LIN {X 0.120,Y -564.110,Z 895.304,A 0.000,B 0.000,C 90.000,E1 90.630} C_DIS
LIN {X 0.098,Y -564.403,Z 895.296,A 0.000,B 0.000,C 90.000,E1 89.255} C_DIS
LIN {X 0.202,Y -564.749,Z 895.287,A 0.000,B 0.000,C 90.000,E1 87.593} C_DIS
LIN {X -0.113,Y -565.091,Z 895.276,A 0.000,B 0.000,C 90.000,E1 85.698} C_DIS
LIN {X 0.186,Y -565.411,Z 895.265,A 0.000,B 0.000,C 90.000,E1 83.742} C_DIS
LIN {X -0.178,Y -565.787,Z 895.256,A 0.000,B 0.000,C 90.000,E1 82.129} C_DIS
LIN {X -0.129,Y -566.486,Z 895.244,A 0.000,B 0.000,C 90.000,E1 79.926} C_DIS
LIN {X -0.025,Y -567.332,Z 895.233,A 0.000,B 0.000,C 90.000,E1 77.993} C_DIS
LIN {X -0.074,Y -568.104,Z 895.224,A 0.000,B 0.000,C 90.000,E1 76.353} C_DIS
LIN {X -0.157,Y -568.803,Z 895.217,A 0.000,B 0.000,C 90.000,E1 74.991} C_DIS
LIN {X -0.072,Y -569.345,Z 895.209,A 0.000,B 0.000,C 90.000,E1 73.614} C_DIS
LIN {X 0.196,Y -569.893,Z 895.200,A 0.000,B 0.000,C 90.000,E1 71.945} C_DIS
LIN {X -0.062,Y -570.251,Z 895.192,A 0.000,B 0.000,C 90.000,E1 70.604} C_DIS
LIN {X -0.125,Y -570.430,Z 895.186,A 0.000,B 0.000,C 90.000,E1 69.518} C_DIS
LIN {X 0.185,Y -570.675,Z 895.177,A 0.000,B 0.000,C 90.000,E1 67.847} C_DIS
LIN {X -0.023,Y -570.852,Z 895.168,A 0.000,B 0.000,C 90.000,E1 66.230} C_DIS
LIN {X 0.003,Y -570.849,Z 895.159,A 0.000,B 0.000,C 90.000,E1 64.588} C_DIS
LIN {X 0.188,Y -570.834,Z 895.151,A 0.000,B 0.000,C 90.000,E1 63.204} C_DIS
LIN {X 0.111,Y -570.663,Z 895.144,A 0.000,B 0.000,C 90.000,E1 61.847} C_DIS
LIN {X 0.134,Y -570.383,Z 895.135,A 0.000,B 0.000,C 90.000,E1 60.205} C_DIS
LIN {X -0.104,Y -570.148,Z 895.130,A 0.000,B 0.000,C 90.000,E1 59.410} C_DIS
LIN {X -0.109,Y -569.555,Z 895.122,A 0.000,B 0.000,C 90.000,E1 58.043} C_DIS
LIN {X 0.241,Y -568.856,Z 895.116,A 0.000,B 0.000,C 90.000,E1 56.914} C_DIS
LIN {X -0.258,Y -567.926,Z 895.109,A 0.000,B 0.000,C 90.000,E1 55.595} C_DIS
LIN {X -0.100,Y -566.927,Z 895.103,A 0.000,B 0.000,C 90.000,E1 54.482} C_DIS
LIN {X 0.034,Y -565.630,Z 895.097,A 0.000,B 0.000,C 90.000,E1 53.371} C_DIS
LIN {X 0.033,Y -564.176,Z 895.090,A 0.000,B 0.000,C 90.000,E1 52.271} C_DIS
LIN {X 0.017,Y -562.468,Z 895.084,A 0.000,B 0.000,C 90.000,E1 51.170} C_DIS
LIN {X -0.118,Y -561.012,Z 895.080,A 0.000,B 0.000,C 90.000,E1 50.356} C_DIS
LIN {X 0.068,Y -559.958,Z 895.077,A 0.000,B 0.000,C 90.000,E1 49.784} C_DIS
LIN {X 0.265,Y -558.069,Z 895.072,A 0.000,B 0.000,C 90.000,E1 48.933} C_DIS
LIN {X -0.339,Y -555.840,Z 895.067,A 0.000,B 0.000,C 90.000,E1 48.162} C_DIS
LIN {X 0.168,Y -554.282,Z 895.064,A 0.000,B 0.000,C 90.000,E1 47.553} C_DIS
LIN {X -0.050,Y -550.551,Z 895.058,A 0.000,B 0.000,C 90.000,E1 46.458} C_DIS
LIN {X 0.014,Y -548.569,Z 895.055,A 0.000,B 0.000,C 90.000,E1 45.891} C_DIS
LIN {X -0.302,Y -545.345,Z 895.050,A 0.000,B 0.000,C 90.000,E1 45.081} C_DIS
LIN {X 0.297,Y -543.590,Z 895.048,A 0.000,B 0.000,C 90.000,E1 44.595} C_DIS
LIN {X 0.307,Y -541.047,Z 895.045,A 0.000,B 0.000,C 90.000,E1 44.028} C_DIS
LIN {X 0.111,Y -537.475,Z 895.041,A 0.000,B 0.000,C 90.000,E1 43.338} C_DIS
LIN {X 0.076,Y -534.403,Z 895.038,A 0.000,B 0.000,C 90.000,E1 42.771} C_DIS
LIN {X -0.006,Y -529.401,Z 895.033,A 0.000,B 0.000,C 90.000,E1 41.919} C_DIS
LIN {X -0.106,Y -525.825,Z 895.030,A 0.000,B 0.000,C 90.000,E1 41.353} C_DIS
LIN {X -0.036,Y -521.095,Z 895.026,A 0.000,B 0.000,C 90.000,E1 40.620} C_DIS
LIN {X -0.003,Y -515.941,Z 895.022,A 0.000,B 0.000,C 90.000,E1 39.886} C_DIS
LIN {X 0.186,Y -511.587,Z 895.018,A 0.000,B 0.000,C 90.000,E1 39.277} C_DIS
LIN {X 0.019,Y -506.960,Z 895.015,A 0.000,B 0.000,C 90.000,E1 38.705} C_DIS
LIN {X 0.089,Y -503.342,Z 895.013,A 0.000,B 0.000,C 90.000,E1 38.257} C_DIS
LIN {X 0.179,Y -499.586,Z 895.010,A 0.000,B 0.000,C 90.000,E1 37.810} C_DIS
LIN {X 0.195,Y -492.719,Z 895.006,A 0.000,B 0.000,C 90.000,E1 37.076} C_DIS
LIN {X -0.048,Y -486.099,Z 895.002,A 0.000,B 0.000,C 90.000,E1 36.423} C_DIS
LIN {X 0.024,Y -478.868,Z 894.999,A 0.000,B 0.000,C 90.000,E1 35.724} C_DIS
LIN {X -0.152,Y -468.392,Z 894.993,A 0.000,B 0.000,C 90.000,E1 34.818} C_DIS
LIN {X -0.046,Y -457.728,Z 894.988,A 0.000,B 0.000,C 90.000,E1 33.913} C_DIS
LIN {X -0.119,Y -446.886,Z 894.984,A 0.000,B 0.000,C 90.000,E1 33.038} C_DIS
LIN {X -0.220,Y -422.099,Z 894.972,A 0.000,B 0.000,C 90.000,E1 31.003} C_DIS
LIN {X -0.148,Y -402.934,Z 894.962,A 0.000,B 0.000,C 90.000,E1 29.205} C_DIS
LIN {X -0.160,Y -397.406,Z 894.959,A 0.000,B 0.000,C 90.000,E1 28.615} C_DIS
LIN {X -0.033,Y -396.068,Z 894.958,A 0.000,B 0.000,C 90.000,E1 28.437} C_DIS
LIN {X 0.170,Y -393.469,Z 894.956,A 0.000,B 0.000,C 90.000,E1 28.025} C_DIS
LIN {X 0.012,Y -391.329,Z 894.954,A 0.000,B 0.000,C 90.000,E1 27.641} C_DIS
LIN {X 0.213,Y -390.228,Z 894.952,A 0.000,B 0.000,C 90.000,E1 27.257} C_DIS
LIN {X -0.127,Y -389.752,Z 894.951,A 0.000,B 0.000,C 90.000,E1 27.129} C_DIS
LIN {X 0.153,Y -388.920,Z 894.947,A 0.000,B 0.000,C 90.000,E1 26.360} C_DIS
LIN {X -0.159,Y -389.105,Z 894.941,A 0.000,B 0.000,C 90.000,E1 25.335} C_DIS
LIN {X 0.125,Y -390.559,Z 894.929,A 0.000,B 0.000,C 90.000,E1 23.153} C_DIS
LIN {X 0.183,Y -393.294,Z 894.913,A 0.000,B 0.000,C 90.000,E1 20.301} C_DIS
LIN {X -0.158,Y -396.046,Z 894.899,A 0.000,B 0.000,C 90.000,E1 17.873} C_DIS
LIN {X 0.134,Y -398.664,Z 894.887,A 0.000,B 0.000,C 90.000,E1 15.717} C_DIS
LIN {X -0.126,Y -401.845,Z 894.874,A 0.000,B 0.000,C 90.000,E1 13.300} C_DIS
LIN {X 0.013,Y -404.867,Z 894.862,A 0.000,B 0.000,C 90.000,E1 11.186} C_DIS
LIN {X 0.112,Y -409.220,Z 894.847,A 0.000,B 0.000,C 90.000,E1 8.398} C_DIS
LIN {X -0.191,Y -412.772,Z 894.835,A 0.000,B 0.000,C 90.000,E1 6.372} C_DIS
LIN {X -0.050,Y -417.361,Z 894.822,A 0.000,B 0.000,C 90.000,E1 3.955} C_DIS
LIN {X -0.176,Y -423.817,Z 894.805,A 0.000,B 0.000,C 90.000,E1 0.917} C_DIS
LIN {X 0.061,Y -430.517,Z 894.790,A 0.000,B 0.000,C 90.000,E1 358.108} C_DIS
LIN {X 0.041,Y -434.907,Z 894.780,A 0.000,B 0.000,C 90.000,E1 356.445} C_DIS
LIN {X 0.172,Y -436.610,Z 894.778,A 0.000,B 0.000,C 90.000,E1 355.931} C_DIS
LIN {X -0.069,Y -438.647,Z 894.775,A 0.000,B 0.000,C 90.000,E1 355.527} C_DIS
LIN {X -0.021,Y -439.577,Z 894.774,A 0.000,B 0.000,C 90.000,E1 355.355} C_DIS
LIN {X 0.171,Y -443.592,Z 894.771,A 0.000,B 0.000,C 90.000,E1 354.837} C_DIS
LIN {X -0.016,Y -448.155,Z 894.770,A 0.000,B 0.000,C 90.000,E1 354.546} C_DIS
LIN {X -0.174,Y -454.270,Z 894.768,A 0.000,B 0.000,C 90.000,E1 354.261} C_DIS
LIN {X -0.090,Y -465.986,Z 894.765,A 0.000,B 0.000,C 90.000,E1 353.742} C_DIS
LIN {X -0.220,Y -476.042,Z 894.763,A 0.000,B 0.000,C 90.000,E1 353.280} C_DIS
LIN {X 0.196,Y -489.174,Z 894.759,A 0.000,B 0.000,C 90.000,E1 352.534} C_DIS
LIN {X 0.058,Y -500.687,Z 894.755,A 0.000,B 0.000,C 90.000,E1 351.894} C_DIS
LIN {X -0.056,Y -510.296,Z 894.752,A 0.000,B 0.000,C 90.000,E1 351.319} C_DIS
LIN {X 0.161,Y -518.210,Z 894.749,A 0.000,B 0.000,C 90.000,E1 350.792} C_DIS
LIN {X 0.052,Y -524.389,Z 894.747,A 0.000,B 0.000,C 90.000,E1 350.387} C_DIS
LIN {X -0.169,Y -531.951,Z 894.744,A 0.000,B 0.000,C 90.000,E1 349.859} C_DIS
LIN {X -0.188,Y -539.120,Z 894.740,A 0.000,B 0.000,C 90.000,E1 349.275} C_DIS
LIN {X 0.105,Y -546.141,Z 894.737,A 0.000,B 0.000,C 90.000,E1 348.634} C_DIS
LIN {X -0.202,Y -552.674,Z 894.734,A 0.000,B 0.000,C 90.000,E1 348.049} C_DIS
LIN {X 0.059,Y -559.083,Z 894.730,A 0.000,B 0.000,C 90.000,E1 347.353} C_DIS
LIN {X 0.161,Y -562.821,Z 894.728,A 0.000,B 0.000,C 90.000,E1 346.937} C_DIS
LIN {X 0.100,Y -569.807,Z 894.723,A 0.000,B 0.000,C 90.000,E1 346.117} C_DIS
LIN {X 0.165,Y -573.085,Z 894.721,A 0.000,B 0.000,C 90.000,E1 345.700} C_DIS
LIN {X 0.007,Y -581.236,Z 894.715,A 0.000,B 0.000,C 90.000,E1 344.629} C_DIS
LIN {X 0.136,Y -584.162,Z 894.712,A 0.000,B 0.000,C 90.000,E1 344.212} C_DIS
LIN {X 0.037,Y -587.773,Z 894.709,A 0.000,B 0.000,C 90.000,E1 343.685} C_DIS
LIN {X 0.245,Y -594.439,Z 894.703,A 0.000,B 0.000,C 90.000,E1 342.598} C_DIS
LIN {X -0.203,Y -600.473,Z 894.698,A 0.000,B 0.000,C 90.000,E1 341.583} C_DIS
LIN {X -0.148,Y -605.417,Z 894.693,A 0.000,B 0.000,C 90.000,E1 340.659} C_DIS
LIN {X 0.312,Y -610.827,Z 894.687,A 0.000,B 0.000,C 90.000,E1 339.571} C_DIS
LIN {X -0.307,Y -615.935,Z 894.681,A 0.000,B 0.000,C 90.000,E1 338.592} C_DIS
LIN {X -0.074,Y -621.306,Z 894.674,A 0.000,B 0.000,C 90.000,E1 337.411} C_DIS
LIN {X 0.239,Y -625.756,Z 894.669,A 0.000,B 0.000,C 90.000,E1 336.357} C_DIS
LIN {X 0.035,Y -629.902,Z 894.663,A 0.000,B 0.000,C 90.000,E1 335.357} C_DIS
LIN {X -0.088,Y -634.662,Z 894.656,A 0.000,B 0.000,C 90.000,E1 334.101} C_DIS
LIN {X 0.040,Y -637.380,Z 894.652,A 0.000,B 0.000,C 90.000,E1 333.332} C_DIS
LIN {X -0.253,Y -641.552,Z 894.645,A 0.000,B 0.000,C 90.000,E1 332.103} C_DIS
LIN {X -0.170,Y -645.310,Z 894.638,A 0.000,B 0.000,C 90.000,E1 330.845} C_DIS
LIN {X 0.138,Y -648.137,Z 894.632,A 0.000,B 0.000,C 90.000,E1 329.822} C_DIS
LIN {X -0.317,Y -650.867,Z 894.627,A 0.000,B 0.000,C 90.000,E1 328.869} C_DIS
LIN {X -0.266,Y -652.784,Z 894.623,A 0.000,B 0.000,C 90.000,E1 328.122} C_DIS
LIN {X -0.193,Y -654.561,Z 894.619,A 0.000,B 0.000,C 90.000,E1 327.375} C_DIS
LIN {X -0.009,Y -656.691,Z 894.613,A 0.000,B 0.000,C 90.000,E1 326.373} C_DIS
LIN {X 0.017,Y -658.504,Z 894.608,A 0.000,B 0.000,C 90.000,E1 325.388} C_DIS
LIN {X 0.134,Y -659.774,Z 894.604,A 0.000,B 0.000,C 90.000,E1 324.642} C_DIS
LIN {X 0.150,Y -661.487,Z 894.597,A 0.000,B 0.000,C 90.000,E1 323.417} C_DIS
LIN {X 0.201,Y -662.840,Z 894.590,A 0.000,B 0.000,C 90.000,E1 322.190} C_DIS
LIN {X 0.246,Y -664.350,Z 894.582,A 0.000,B 0.000,C 90.000,E1 320.723} C_DIS
LIN {X 0.263,Y -665.356,Z 894.577,A 0.000,B 0.000,C 90.000,E1 319.747} C_DIS
LIN {X -0.165,Y -667.034,Z 894.567,A 0.000,B 0.000,C 90.000,E1 318.081} C_DIS
LIN {X -0.120,Y -668.650,Z 894.559,A 0.000,B 0.000,C 90.000,E1 316.620} C_DIS
LIN {X -0.091,Y -669.668,Z 894.554,A 0.000,B 0.000,C 90.000,E1 315.648} C_DIS
LIN {X -0.045,Y -670.523,Z 894.548,A 0.000,B 0.000,C 90.000,E1 314.676} C_DIS
LIN {X -0.388,Y -672.416,Z 894.537,A 0.000,B 0.000,C 90.000,E1 312.771} C_DIS
LIN {X -0.235,Y -673.775,Z 894.529,A 0.000,B 0.000,C 90.000,E1 311.310} C_DIS
LIN {X 0.041,Y -675.168,Z 894.520,A 0.000,B 0.000,C 90.000,E1 309.600} C_DIS
LIN {X 0.214,Y -676.187,Z 894.513,A 0.000,B 0.000,C 90.000,E1 308.382} C_DIS
LIN {X 0.103,Y -677.207,Z 894.505,A 0.000,B 0.000,C 90.000,E1 306.950} C_DIS
LIN {X 0.013,Y -678.045,Z 894.499,A 0.000,B 0.000,C 90.000,E1 305.758} C_DIS
LIN {X 0.102,Y -678.945,Z 894.489,A 0.000,B 0.000,C 90.000,E1 304.072} C_DIS
LIN {X -0.178,Y -679.944,Z 894.480,A 0.000,B 0.000,C 90.000,E1 302.418} C_DIS
LIN {X 0.125,Y -681.193,Z 894.471,A 0.000,B 0.000,C 90.000,E1 300.718} C_DIS
LIN {X -0.008,Y -683.717,Z 894.456,A 0.000,B 0.000,C 90.000,E1 298.103} C_DIS
LIN {X 0.198,Y -686.005,Z 894.446,A 0.000,B 0.000,C 90.000,E1 296.181} C_DIS
LIN {X 0.005,Y -687.787,Z 894.438,A 0.000,B 0.000,C 90.000,E1 294.771} C_DIS
LIN {X -0.002,Y -688.728,Z 894.432,A 0.000,B 0.000,C 90.000,E1 293.823} C_DIS
LIN {X -0.051,Y -688.945,Z 894.431,A 0.000,B 0.000,C 90.000,E1 293.590} C_DIS
LIN {X -0.230,Y -688.968,Z 894.428,A 0.000,B 0.000,C 90.000,E1 293.131} C_DIS
LIN {X -0.272,Y -688.919,Z 894.427,A 0.000,B 0.000,C 90.000,E1 292.898} C_DIS
LIN {X 0.176,Y -687.942,Z 894.424,A 0.000,B 0.000,C 90.000,E1 292.386} C_DIS
LIN {X 0.137,Y -687.332,Z 894.423,A 0.000,B 0.000,C 90.000,E1 292.153} C_DIS
LIN {X 0.246,Y -686.760,Z 894.423,A 0.000,B 0.000,C 90.000,E1 292.025} C_DIS
LIN {X 0.207,Y -684.913,Z 894.421,A 0.000,B 0.000,C 90.000,E1 291.791} C_DIS
LIN {X -0.116,Y -681.619,Z 894.419,A 0.000,B 0.000,C 90.000,E1 291.461} C_DIS
LIN {X -0.266,Y -680.064,Z 894.419,A 0.000,B 0.000,C 90.000,E1 291.354} C_DIS
LIN {X -0.166,Y -677.426,Z 894.418,A 0.000,B 0.000,C 90.000,E1 291.227} C_DIS
LIN {X -0.319,Y -668.621,Z 894.416,A 0.000,B 0.000,C 90.000,E1 290.918} C_DIS
LIN {X -0.218,Y -666.510,Z 894.416,A 0.000,B 0.000,C 90.000,E1 290.844} C_DIS
LIN {X 0.243,Y -662.821,Z 894.415,A 0.000,B 0.000,C 90.000,E1 290.663} C_DIS
LIN {X 0.012,Y -658.681,Z 894.414,A 0.000,B 0.000,C 90.000,E1 290.482} C_DIS
LIN {X -0.045,Y -658.599,Z 894.414,A 0.000,B 0.000,C 90.000,E1 290.482} C_DIS
LIN {X 0.119,Y -658.032,Z 894.413,A 0.000,B 0.000,C 90.000,E1 290.375} C_DIS
LIN {X 0.063,Y -658.020,Z 894.413,A 0.000,B 0.000,C 90.000,E1 290.375} C_DIS
LIN {X 0.000,Y -658.050,Z 894.412,A 0.000,B 0.000,C 90.000,E1 290.120} C_DIS
LIN {X 0.012,Y -659.624,Z 894.409,A 0.000,B 0.000,C 90.000,E1 289.631} C_DIS
LIN {X -0.105,Y -663.109,Z 894.405,A 0.000,B 0.000,C 90.000,E1 288.906} C_DIS
LIN {X -0.124,Y -667.590,Z 894.400,A 0.000,B 0.000,C 90.000,E1 288.055} C_DIS
LIN {X -0.289,Y -670.016,Z 894.398,A 0.000,B 0.000,C 90.000,E1 287.583} C_DIS
LIN {X -0.239,Y -672.299,Z 894.395,A 0.000,B 0.000,C 90.000,E1 287.094} C_DIS
LIN {X 0.405,Y -675.179,Z 894.391,A 0.000,B 0.000,C 90.000,E1 286.315} C_DIS
LIN {X 0.295,Y -676.749,Z 894.388,A 0.000,B 0.000,C 90.000,E1 285.843} C_DIS
LIN {X 0.153,Y -678.656,Z 894.384,A 0.000,B 0.000,C 90.000,E1 285.134} C_DIS
LIN {X 0.033,Y -680.242,Z 894.380,A 0.000,B 0.000,C 90.000,E1 284.426} C_DIS
LIN {X -0.103,Y -681.996,Z 894.375,A 0.000,B 0.000,C 90.000,E1 283.480} C_DIS
LIN {X -0.220,Y -683.291,Z 894.370,A 0.000,B 0.000,C 90.000,E1 282.535} C_DIS
LIN {X -0.304,Y -683.893,Z 894.366,A 0.000,B 0.000,C 90.000,E1 281.827} C_DIS
LIN {X 0.309,Y -684.056,Z 894.363,A 0.000,B 0.000,C 90.000,E1 281.299} C_DIS
LIN {X 0.094,Y -683.745,Z 894.359,A 0.000,B 0.000,C 90.000,E1 280.602} C_DIS
LIN {X -0.089,Y -683.310,Z 894.356,A 0.000,B 0.000,C 90.000,E1 280.141} C_DIS
LIN {X -0.155,Y -682.489,Z 894.354,A 0.000,B 0.000,C 90.000,E1 279.670} C_DIS
LIN {X 0.290,Y -680.648,Z 894.350,A 0.000,B 0.000,C 90.000,E1 278.916} C_DIS
LIN {X 0.096,Y -679.078,Z 894.347,A 0.000,B 0.000,C 90.000,E1 278.454} C_DIS
LIN {X -0.104,Y -677.225,Z 894.344,A 0.000,B 0.000,C 90.000,E1 277.992} C_DIS
LIN {X -0.315,Y -675.040,Z 894.342,A 0.000,B 0.000,C 90.000,E1 277.530} C_DIS
LIN {X 0.134,Y -672.040,Z 894.338,A 0.000,B 0.000,C 90.000,E1 276.891} C_DIS
LIN {X -0.197,Y -668.558,Z 894.335,A 0.000,B 0.000,C 90.000,E1 276.315} C_DIS
LIN {X 0.198,Y -665.547,Z 894.332,A 0.000,B 0.000,C 90.000,E1 275.796} C_DIS
LIN {X -0.092,Y -662.135,Z 894.330,A 0.000,B 0.000,C 90.000,E1 275.334} C_DIS
LIN {X 0.156,Y -657.183,Z 894.326,A 0.000,B 0.000,C 90.000,E1 274.702} C_DIS
LIN {X -0.237,Y -652.744,Z 894.323,A 0.000,B 0.000,C 90.000,E1 274.245} C_DIS
LIN {X 0.008,Y -646.618,Z 894.320,A 0.000,B 0.000,C 90.000,E1 273.612} C_DIS
LIN {X -0.163,Y -641.381,Z 894.318,A 0.000,B 0.000,C 90.000,E1 273.154} C_DIS
LIN {X -0.137,Y -635.889,Z 894.315,A 0.000,B 0.000,C 90.000,E1 272.694} C_DIS
LIN {X 0.137,Y -630.196,Z 894.313,A 0.000,B 0.000,C 90.000,E1 272.236} C_DIS
LIN {X 0.048,Y -624.229,Z 894.310,A 0.000,B 0.000,C 90.000,E1 271.835} C_DIS
LIN {X 0.189,Y -617.797,Z 894.308,A 0.000,B 0.000,C 90.000,E1 271.432} C_DIS
LIN {X 0.054,Y -611.186,Z 894.306,A 0.000,B 0.000,C 90.000,E1 271.088} C_DIS
LIN {X 0.208,Y -604.430,Z 894.304,A 0.000,B 0.000,C 90.000,E1 270.745} C_DIS
LIN {X 0.020,Y -597.438,Z 894.303,A 0.000,B 0.000,C 90.000,E1 270.458} C_DIS
LIN {X 0.131,Y -590.087,Z 894.301,A 0.000,B 0.000,C 90.000,E1 270.172} C_DIS
LIN {X 0.021,Y -584.559,Z 894.300,A 0.000,B 0.000,C 90.000,E1 270.000} C_DIS
LIN {X -0.267,Y -576.802,Z 894.299,A 0.000,B 0.000,C 90.000,E1 269.828} C_DIS
LIN {X 0.265,Y -570.875,Z 894.298,A 0.000,B 0.000,C 90.000,E1 269.656} C_DIS
LIN {X -0.150,Y -563.574,Z 894.298,A 0.000,B 0.000,C 90.000,E1 269.599} C_DIS
LIN {X 0.188,Y -553.327,Z 894.297,A 0.000,B 0.000,C 90.000,E1 269.484} C_DIS
LIN {X -0.197,Y -551.584,Z 894.297,A 0.000,B 0.000,C 90.000,E1 269.484} C_DIS
LIN {X -0.086,Y -550.159,Z 894.297,A 0.000,B 0.000,C 90.000,E1 269.427} C_DIS
LIN {X -0.119,Y -550.110,Z 894.297,A 0.000,B 0.000,C 90.000,E1 269.427} C_DIS
LIN {X -0.121,Y -547.333,Z 894.295,A 0.000,B 0.000,C 90.000,E1 269.083} C_DIS
LIN {X 0.138,Y -545.221,Z 894.293,A 0.000,B 0.000,C 90.000,E1 268.740} C_DIS
LIN {X -0.030,Y -544.632,Z 894.292,A 0.000,B 0.000,C 90.000,E1 268.511} C_DIS
LIN {X 0.233,Y -542.363,Z 894.281,A 0.000,B 0.000,C 90.000,E1 266.502} C_DIS
LIN {X -0.035,Y -540.700,Z 894.268,A 0.000,B 0.000,C 90.000,E1 264.261} C_DIS
LIN {X 0.104,Y -539.976,Z 894.262,A 0.000,B 0.000,C 90.000,E1 263.109} C_DIS
LIN {X -0.235,Y -539.038,Z 894.255,A 0.000,B 0.000,C 90.000,E1 262.008} C_DIS
LIN {X 0.017,Y -537.639,Z 894.248,A 0.000,B 0.000,C 90.000,E1 260.557} C_DIS
LIN {X -0.170,Y -535.598,Z 894.237,A 0.000,B 0.000,C 90.000,E1 258.578} C_DIS
LIN {X 0.054,Y -534.335,Z 894.230,A 0.000,B 0.000,C 90.000,E1 257.409} C_DIS
LIN {X -0.142,Y -532.924,Z 894.224,A 0.000,B 0.000,C 90.000,E1 256.284} C_DIS
LIN {X -0.278,Y -530.722,Z 894.214,A 0.000,B 0.000,C 90.000,E1 254.574} C_DIS
LIN {X 0.153,Y -528.989,Z 894.206,A 0.000,B 0.000,C 90.000,E1 253.087} C_DIS
LIN {X -0.295,Y -526.862,Z 894.197,A 0.000,B 0.000,C 90.000,E1 251.402} C_DIS
LIN {X -0.111,Y -525.070,Z 894.188,A 0.000,B 0.000,C 90.000,E1 249.934} C_DIS
LIN {X 0.206,Y -522.700,Z 894.179,A 0.000,B 0.000,C 90.000,E1 248.156} C_DIS
LIN {X 0.151,Y -521.029,Z 894.172,A 0.000,B 0.000,C 90.000,E1 246.997} C_DIS
LIN {X 0.002,Y -519.307,Z 894.166,A 0.000,B 0.000,C 90.000,E1 245.845} C_DIS
LIN {X 0.117,Y -516.616,Z 894.156,A 0.000,B 0.000,C 90.000,E1 244.076} C_DIS
LIN {X -0.076,Y -514.743,Z 894.150,A 0.000,B 0.000,C 90.000,E1 242.922} C_DIS
LIN {X 0.147,Y -511.683,Z 894.140,A 0.000,B 0.000,C 90.000,E1 241.129} C_DIS
LIN {X -0.025,Y -508.052,Z 894.128,A 0.000,B 0.000,C 90.000,E1 239.076} C_DIS
LIN {X 0.036,Y -505.434,Z 894.120,A 0.000,B 0.000,C 90.000,E1 237.582} C_DIS
LIN {X 0.163,Y -503.077,Z 894.113,A 0.000,B 0.000,C 90.000,E1 236.373} C_DIS
LIN {X -0.183,Y -501.160,Z 894.108,A 0.000,B 0.000,C 90.000,E1 235.515} C_DIS
LIN {X -0.237,Y -496.229,Z 894.097,A 0.000,B 0.000,C 90.000,E1 233.417} C_DIS
LIN {X -0.234,Y -492.905,Z 894.088,A 0.000,B 0.000,C 90.000,E1 231.904} C_DIS
LIN {X -0.152,Y -488.727,Z 894.078,A 0.000,B 0.000,C 90.000,E1 230.070} C_DIS
LIN {X -0.044,Y -485.396,Z 894.070,A 0.000,B 0.000,C 90.000,E1 228.528} C_DIS
LIN {X -0.064,Y -480.505,Z 894.058,A 0.000,B 0.000,C 90.000,E1 226.377} C_DIS
LIN {X -0.246,Y -477.730,Z 894.051,A 0.000,B 0.000,C 90.000,E1 225.162} C_DIS
LIN {X -0.018,Y -474.165,Z 894.042,A 0.000,B 0.000,C 90.000,E1 223.581} C_DIS
LIN {X 0.278,Y -472.129,Z 894.037,A 0.000,B 0.000,C 90.000,E1 222.609} C_DIS
LIN {X -0.162,Y -467.863,Z 894.026,A 0.000,B 0.000,C 90.000,E1 220.782} C_DIS
LIN {X -0.044,Y -463.817,Z 894.016,A 0.000,B 0.000,C 90.000,E1 218.874} C_DIS
LIN {X -0.022,Y -461.180,Z 894.009,A 0.000,B 0.000,C 90.000,E1 217.604} C_DIS
LIN {X -0.017,Y -457.786,Z 894.000,A 0.000,B 0.000,C 90.000,E1 216.011} C_DIS
LIN {X -0.160,Y -453.037,Z 893.988,A 0.000,B 0.000,C 90.000,E1 213.785} C_DIS
LIN {X -0.063,Y -448.213,Z 893.975,A 0.000,B 0.000,C 90.000,E1 211.514} C_DIS
LIN {X 0.029,Y -442.494,Z 893.961,A 0.000,B 0.000,C 90.000,E1 208.899} C_DIS
LIN {X 0.053,Y -438.840,Z 893.952,A 0.000,B 0.000,C 90.000,E1 207.257} C_DIS
LIN {X 0.012,Y -434.522,Z 893.941,A 0.000,B 0.000,C 90.000,E1 205.283} C_DIS
LIN {X -0.124,Y -430.981,Z 893.931,A 0.000,B 0.000,C 90.000,E1 203.643} C_DIS
LIN {X 0.055,Y -426.049,Z 893.918,A 0.000,B 0.000,C 90.000,E1 201.280} C_DIS
LIN {X 0.002,Y -421.838,Z 893.907,A 0.000,B 0.000,C 90.000,E1 199.268} C_DIS
LIN {X 0.114,Y -417.764,Z 893.896,A 0.000,B 0.000,C 90.000,E1 197.221} C_DIS
LIN {X -0.140,Y -414.218,Z 893.886,A 0.000,B 0.000,C 90.000,E1 195.552} C_DIS
LIN {X -0.038,Y -410.197,Z 893.875,A 0.000,B 0.000,C 90.000,E1 193.480} C_DIS
LIN {X -0.146,Y -406.948,Z 893.865,A 0.000,B 0.000,C 90.000,E1 191.771} C_DIS
LIN {X -0.019,Y -404.219,Z 893.858,A 0.000,B 0.000,C 90.000,E1 190.366} C_DIS
LIN {X -0.027,Y -399.966,Z 893.846,A 0.000,B 0.000,C 90.000,E1 188.276} C_DIS
LIN {X 0.150,Y -395.831,Z 893.834,A 0.000,B 0.000,C 90.000,E1 186.144} C_DIS
LIN {X -0.165,Y -392.075,Z 893.823,A 0.000,B 0.000,C 90.000,E1 184.069} C_DIS
LIN {X 0.054,Y -388.090,Z 893.809,A 0.000,B 0.000,C 90.000,E1 181.547} C_DIS
LIN {X -0.035,Y -385.413,Z 893.799,A 0.000,B 0.000,C 90.000,E1 179.771} C_DIS
LIN {X 0.102,Y -382.098,Z 893.787,A 0.000,B 0.000,C 90.000,E1 177.593} C_DIS
LIN {X 0.096,Y -376.948,Z 893.767,A 0.000,B 0.000,C 90.000,E1 173.970} C_DIS
LIN {X 0.109,Y -376.021,Z 893.761,A 0.000,B 0.000,C 90.000,E1 172.875} C_DIS
LIN {X -0.157,Y -375.553,Z 893.757,A 0.000,B 0.000,C 90.000,E1 172.186} C_DIS
LIN {X -0.031,Y -375.411,Z 893.751,A 0.000,B 0.000,C 90.000,E1 171.254} C_DIS
LIN {X 0.035,Y -375.991,Z 893.746,A 0.000,B 0.000,C 90.000,E1 170.330} C_DIS
LIN {X -0.183,Y -376.944,Z 893.742,A 0.000,B 0.000,C 90.000,E1 169.634} C_DIS
LIN {X 0.051,Y -378.605,Z 893.738,A 0.000,B 0.000,C 90.000,E1 168.870} C_DIS
LIN {X -0.052,Y -379.726,Z 893.736,A 0.000,B 0.000,C 90.000,E1 168.522} C_DIS
LIN {X -0.093,Y -381.690,Z 893.734,A 0.000,B 0.000,C 90.000,E1 168.117} C_DIS
LIN {X -0.102,Y -382.783,Z 893.733,A 0.000,B 0.000,C 90.000,E1 167.937} C_DIS
LIN {X 0.003,Y -385.840,Z 893.731,A 0.000,B 0.000,C 90.000,E1 167.521} C_DIS
LIN {X 0.142,Y -390.433,Z 893.728,A 0.000,B 0.000,C 90.000,E1 166.992} C_DIS
LIN {X 0.099,Y -397.294,Z 893.725,A 0.000,B 0.000,C 90.000,E1 166.464} C_DIS
LIN {X -0.104,Y -412.743,Z 893.720,A 0.000,B 0.000,C 90.000,E1 165.574} C_DIS
LIN {X -0.195,Y -417.736,Z 893.718,A 0.000,B 0.000,C 90.000,E1 165.283} C_DIS
LIN {X -0.188,Y -427.254,Z 893.715,A 0.000,B 0.000,C 90.000,E1 164.629} C_DIS
LIN {X -0.054,Y -435.214,Z 893.711,A 0.000,B 0.000,C 90.000,E1 164.031} C_DIS
LIN {X -0.159,Y -441.348,Z 893.709,A 0.000,B 0.000,C 90.000,E1 163.559} C_DIS
LIN {X 0.253,Y -451.904,Z 893.704,A 0.000,B 0.000,C 90.000,E1 162.598} C_DIS
LIN {X 0.175,Y -460.367,Z 893.699,A 0.000,B 0.000,C 90.000,E1 161.819} C_DIS
LIN {X -0.038,Y -470.264,Z 893.694,A 0.000,B 0.000,C 90.000,E1 160.859} C_DIS
LIN {X 0.182,Y -478.294,Z 893.689,A 0.000,B 0.000,C 90.000,E1 159.934} C_DIS
LIN {X -0.011,Y -482.197,Z 893.686,A 0.000,B 0.000,C 90.000,E1 159.518} C_DIS
LIN {X 0.028,Y -487.264,Z 893.683,A 0.000,B 0.000,C 90.000,E1 158.901} C_DIS
LIN {X -0.142,Y -493.314,Z 893.679,A 0.000,B 0.000,C 90.000,E1 158.156} C_DIS
LIN {X -0.055,Y -497.804,Z 893.675,A 0.000,B 0.000,C 90.000,E1 157.539} C_DIS
LIN {X 0.002,Y -500.076,Z 893.674,A 0.000,B 0.000,C 90.000,E1 157.230} C_DIS
LIN {X 0.033,Y -507.628,Z 893.668,A 0.000,B 0.000,C 90.000,E1 156.177} C_DIS
LIN {X 0.200,Y -515.963,Z 893.661,A 0.000,B 0.000,C 90.000,E1 154.973} C_DIS
LIN {X -0.132,Y -524.848,Z 893.654,A 0.000,B 0.000,C 90.000,E1 153.691} C_DIS
LIN {X 0.145,Y -533.305,Z 893.647,A 0.000,B 0.000,C 90.000,E1 152.359} C_DIS
LIN {X 0.154,Y -537.634,Z 893.643,A 0.000,B 0.000,C 90.000,E1 151.641} C_DIS
LIN {X -0.136,Y -540.846,Z 893.639,A 0.000,B 0.000,C 90.000,E1 151.101} C_DIS
LIN {X 0.158,Y -546.622,Z 893.634,A 0.000,B 0.000,C 90.000,E1 150.078} C_DIS
LIN {X -0.152,Y -551.883,Z 893.628,A 0.000,B 0.000,C 90.000,E1 149.125} C_DIS
LIN {X -0.097,Y -556.401,Z 893.624,A 0.000,B 0.000,C 90.000,E1 148.280} C_DIS
LIN {X -0.104,Y -564.443,Z 893.615,A 0.000,B 0.000,C 90.000,E1 146.755} C_DIS
LIN {X -0.069,Y -570.510,Z 893.608,A 0.000,B 0.000,C 90.000,E1 145.515} C_DIS
LIN {X 0.205,Y -577.543,Z 893.600,A 0.000,B 0.000,C 90.000,E1 143.989} C_DIS
LIN {X -0.121,Y -581.315,Z 893.596,A 0.000,B 0.000,C 90.000,E1 143.210} C_DIS
LIN {X 0.222,Y -587.803,Z 893.587,A 0.000,B 0.000,C 90.000,E1 141.698} C_DIS
LIN {X -0.186,Y -591.944,Z 893.582,A 0.000,B 0.000,C 90.000,E1 140.803} C_DIS
LIN {X -0.251,Y -596.519,Z 893.576,A 0.000,B 0.000,C 90.000,E1 139.747} C_DIS
LIN {X -0.228,Y -603.362,Z 893.568,A 0.000,B 0.000,C 90.000,E1 138.162} C_DIS
LIN {X 0.085,Y -609.195,Z 893.560,A 0.000,B 0.000,C 90.000,E1 136.824} C_DIS
LIN {X -0.367,Y -614.975,Z 893.553,A 0.000,B 0.000,C 90.000,E1 135.567} C_DIS
LIN {X 0.014,Y -618.506,Z 893.549,A 0.000,B 0.000,C 90.000,E1 134.757} C_DIS
LIN {X 0.143,Y -624.024,Z 893.542,A 0.000,B 0.000,C 90.000,E1 133.461} C_DIS
LIN {X 0.057,Y -628.482,Z 893.536,A 0.000,B 0.000,C 90.000,E1 132.447} C_DIS
LIN {X 0.272,Y -634.802,Z 893.527,A 0.000,B 0.000,C 90.000,E1 130.906} C_DIS
LIN {X 0.012,Y -637.991,Z 893.523,A 0.000,B 0.000,C 90.000,E1 130.172} C_DIS
LIN {X -0.310,Y -641.938,Z 893.518,A 0.000,B 0.000,C 90.000,E1 129.197} C_DIS
LIN {X 0.249,Y -647.670,Z 893.509,A 0.000,B 0.000,C 90.000,E1 127.649} C_DIS
LIN {X -0.277,Y -650.525,Z 893.505,A 0.000,B 0.000,C 90.000,E1 126.950} C_DIS
LIN {X 0.130,Y -655.044,Z 893.498,A 0.000,B 0.000,C 90.000,E1 125.678} C_DIS
LIN {X 0.073,Y -659.314,Z 893.492,A 0.000,B 0.000,C 90.000,E1 124.452} C_DIS
LIN {X -0.120,Y -663.291,Z 893.485,A 0.000,B 0.000,C 90.000,E1 123.245} C_DIS
LIN {X -0.013,Y -666.047,Z 893.479,A 0.000,B 0.000,C 90.000,E1 122.260} C_DIS
LIN {X -0.163,Y -667.978,Z 893.475,A 0.000,B 0.000,C 90.000,E1 121.544} C_DIS
LIN {X 0.060,Y -669.634,Z 893.471,A 0.000,B 0.000,C 90.000,E1 120.797} C_DIS
LIN {X 0.120,Y -671.498,Z 893.466,A 0.000,B 0.000,C 90.000,E1 119.823} C_DIS
LIN {X -0.047,Y -673.122,Z 893.460,A 0.000,B 0.000,C 90.000,E1 118.871} C_DIS
LIN {X -0.178,Y -675.286,Z 893.452,A 0.000,B 0.000,C 90.000,E1 117.436} C_DIS
LIN {X -0.352,Y -676.375,Z 893.447,A 0.000,B 0.000,C 90.000,E1 116.488} C_DIS
LIN {X -0.314,Y -677.222,Z 893.440,A 0.000,B 0.000,C 90.000,E1 115.283} C_DIS
LIN {X 0.256,Y -677.417,Z 893.436,A 0.000,B 0.000,C 90.000,E1 114.515} C_DIS
LIN {X -0.263,Y -677.374,Z 893.434,A 0.000,B 0.000,C 90.000,E1 114.079} C_DIS
LIN {X 0.029,Y -676.832,Z 893.430,A 0.000,B 0.000,C 90.000,E1 113.334} C_DIS
LIN {X 0.134,Y -675.626,Z 893.427,A 0.000,B 0.000,C 90.000,E1 112.845} C_DIS
LIN {X -0.307,Y -674.768,Z 893.426,A 0.000,B 0.000,C 90.000,E1 112.642} C_DIS
LIN {X -0.215,Y -671.238,Z 893.423,A 0.000,B 0.000,C 90.000,E1 112.153} C_DIS
LIN {X -0.131,Y -670.245,Z 893.422,A 0.000,B 0.000,C 90.000,E1 112.025} C_DIS
LIN {X -0.050,Y -668.746,Z 893.422,A 0.000,B 0.000,C 90.000,E1 111.897} C_DIS
LIN {X 0.155,Y -664.780,Z 893.420,A 0.000,B 0.000,C 90.000,E1 111.663} C_DIS
LIN {X -0.233,Y -663.050,Z 893.420,A 0.000,B 0.000,C 90.000,E1 111.589} C_DIS
LIN {X 0.164,Y -660.961,Z 893.419,A 0.000,B 0.000,C 90.000,E1 111.461} C_DIS
LIN {X -0.178,Y -654.692,Z 893.418,A 0.000,B 0.000,C 90.000,E1 111.280} C_DIS
LIN {X -0.074,Y -649.144,Z 893.418,A 0.000,B 0.000,C 90.000,E1 111.153} C_DIS
LIN {X 0.206,Y -631.569,Z 893.416,A 0.000,B 0.000,C 90.000,E1 110.791} C_DIS
LIN {X 0.144,Y -618.694,Z 893.414,A 0.000,B 0.000,C 90.000,E1 110.482} C_DIS
LIN {X 0.122,Y -611.369,Z 893.413,A 0.000,B 0.000,C 90.000,E1 110.248} C_DIS
LIN {X -0.020,Y -603.984,Z 893.411,A 0.000,B 0.000,C 90.000,E1 109.939} C_DIS
LIN {X 0.328,Y -595.029,Z 893.408,A 0.000,B 0.000,C 90.000,E1 109.450} C_DIS
LIN {X 0.187,Y -587.129,Z 893.406,A 0.000,B 0.000,C 90.000,E1 109.033} C_DIS
LIN {X 0.161,Y -582.165,Z 893.404,A 0.000,B 0.000,C 90.000,E1 108.779} C_DIS
LIN {X -0.053,Y -579.056,Z 893.404,A 0.000,B 0.000,C 90.000,E1 108.652} C_DIS
LIN {X -0.049,Y -569.835,Z 893.402,A 0.000,B 0.000,C 90.000,E1 108.290} C_DIS
LIN {X 0.329,Y -564.369,Z 893.401,A 0.000,B 0.000,C 90.000,E1 108.055} C_DIS
LIN {X -0.202,Y -561.827,Z 893.400,A 0.000,B 0.000,C 90.000,E1 108.000} C_DIS
LIN {X 0.219,Y -558.316,Z 893.399,A 0.000,B 0.000,C 90.000,E1 107.764} C_DIS
LIN {X 0.173,Y -558.259,Z 893.399,A 0.000,B 0.000,C 90.000,E1 107.764} C_DIS
LIN {X 0.139,Y -556.771,Z 893.398,A 0.000,B 0.000,C 90.000,E1 107.528} C_DIS
LIN {X -0.054,Y -556.111,Z 893.395,A 0.000,B 0.000,C 90.000,E1 107.166} C_DIS
LIN {X 0.260,Y -555.971,Z 893.393,A 0.000,B 0.000,C 90.000,E1 106.677} C_DIS
LIN {X 0.096,Y -556.823,Z 893.379,A 0.000,B 0.000,C 90.000,E1 104.189} C_DIS
LIN {X -0.167,Y -558.196,Z 893.365,A 0.000,B 0.000,C 90.000,E1 101.715} C_DIS
LIN {X 0.285,Y -559.579,Z 893.354,A 0.000,B 0.000,C 90.000,E1 99.726} C_DIS
LIN {X -0.270,Y -560.613,Z 893.347,A 0.000,B 0.000,C 90.000,E1 98.398} C_DIS
LIN {X 0.048,Y -561.773,Z 893.336,A 0.000,B 0.000,C 90.000,E1 96.429} C_DIS
LIN {X 0.171,Y -562.673,Z 893.327,A 0.000,B 0.000,C 90.000,E1 94.759} C_DIS
LIN {X 0.130,Y -563.281,Z 893.319,A 0.000,B 0.000,C 90.000,E1 93.383} C_DIS
LIN {X 0.235,Y -563.905,Z 893.310,A 0.000,B 0.000,C 90.000,E1 91.718} C_DIS
LIN {X 0.097,Y -564.266,Z 893.304,A 0.000,B 0.000,C 90.000,E1 90.630} C_DIS
LIN {X 0.078,Y -564.568,Z 893.296,A 0.000,B 0.000,C 90.000,E1 89.255} C_DIS
LIN {X 0.186,Y -564.910,Z 893.287,A 0.000,B 0.000,C 90.000,E1 87.593} C_DIS
LIN {X -0.125,Y -565.219,Z 893.276,A 0.000,B 0.000,C 90.000,E1 85.698} C_DIS
LIN {X -0.289,Y -565.622,Z 893.264,A 0.000,B 0.000,C 90.000,E1 83.514} C_DIS
LIN {X -0.019,Y -565.993,Z 893.255,A 0.000,B 0.000,C 90.000,E1 81.837} C_DIS
LIN {X 0.041,Y -566.744,Z 893.242,A 0.000,B 0.000,C 90.000,E1 79.634} C_DIS
LIN {X 0.154,Y -567.602,Z 893.232,A 0.000,B 0.000,C 90.000,E1 77.701} C_DIS
LIN {X 0.106,Y -568.367,Z 893.223,A 0.000,B 0.000,C 90.000,E1 76.061} C_DIS
LIN {X 0.025,Y -569.030,Z 893.215,A 0.000,B 0.000,C 90.000,E1 74.700} C_DIS
LIN {X 0.110,Y -569.565,Z 893.207,A 0.000,B 0.000,C 90.000,E1 73.323} C_DIS
LIN {X 0.173,Y -570.151,Z 893.197,A 0.000,B 0.000,C 90.000,E1 71.402} C_DIS
LIN {X -0.081,Y -570.454,Z 893.189,A 0.000,B 0.000,C 90.000,E1 70.061} C_DIS
LIN {X -0.154,Y -570.713,Z 893.179,A 0.000,B 0.000,C 90.000,E1 68.156} C_DIS
LIN {X -0.007,Y -570.883,Z 893.168,A 0.000,B 0.000,C 90.000,E1 66.230} C_DIS
LIN {X 0.019,Y -570.880,Z 893.159,A 0.000,B 0.000,C 90.000,E1 64.588} C_DIS
LIN {X -0.305,Y -570.842,Z 893.151,A 0.000,B 0.000,C 90.000,E1 63.256} C_DIS
LIN {X 0.128,Y -570.664,Z 893.144,A 0.000,B 0.000,C 90.000,E1 61.847} C_DIS
LIN {X 0.150,Y -570.358,Z 893.135,A 0.000,B 0.000,C 90.000,E1 60.205} C_DIS
LIN {X -0.088,Y -570.104,Z 893.130,A 0.000,B 0.000,C 90.000,E1 59.410} C_DIS
LIN {X -0.276,Y -569.347,Z 893.121,A 0.000,B 0.000,C 90.000,E1 57.788} C_DIS
LIN {X -0.168,Y -568.211,Z 893.112,A 0.000,B 0.000,C 90.000,E1 56.135} C_DIS
LIN {X -0.123,Y -567.549,Z 893.107,A 0.000,B 0.000,C 90.000,E1 55.308} C_DIS
LIN {X -0.089,Y -566.777,Z 893.103,A 0.000,B 0.000,C 90.000,E1 54.482} C_DIS
LIN {X -0.296,Y -565.072,Z 893.095,A 0.000,B 0.000,C 90.000,E1 53.130} C_DIS
LIN {X 0.040,Y -563.969,Z 893.090,A 0.000,B 0.000,C 90.000,E1 52.271} C_DIS
LIN {X -0.082,Y -562.703,Z 893.086,A 0.000,B 0.000,C 90.000,E1 51.457} C_DIS
LIN {X -0.213,Y -561.275,Z 893.081,A 0.000,B 0.000,C 90.000,E1 50.642} C_DIS
LIN {X 0.067,Y -559.647,Z 893.077,A 0.000,B 0.000,C 90.000,E1 49.784} C_DIS
LIN {X 0.261,Y -557.718,Z 893.072,A 0.000,B 0.000,C 90.000,E1 48.933} C_DIS
LIN {X -0.004,Y -556.269,Z 893.069,A 0.000,B 0.000,C 90.000,E1 48.405} C_DIS
LIN {X 0.156,Y -553.853,Z 893.064,A 0.000,B 0.000,C 90.000,E1 47.553} C_DIS
LIN {X -0.067,Y -550.074,Z 893.058,A 0.000,B 0.000,C 90.000,E1 46.458} C_DIS
LIN {X -0.007,Y -548.047,Z 893.055,A 0.000,B 0.000,C 90.000,E1 45.891} C_DIS
LIN {X 0.040,Y -545.902,Z 893.052,A 0.000,B 0.000,C 90.000,E1 45.324} C_DIS
LIN {X 0.072,Y -543.623,Z 893.049,A 0.000,B 0.000,C 90.000,E1 44.757} C_DIS
LIN {X 0.274,Y -540.396,Z 893.045,A 0.000,B 0.000,C 90.000,E1 44.028} C_DIS
LIN {X 0.259,Y -537.561,Z 893.042,A 0.000,B 0.000,C 90.000,E1 43.461} C_DIS
LIN {X -0.144,Y -534.499,Z 893.038,A 0.000,B 0.000,C 90.000,E1 42.933} C_DIS
LIN {X -0.033,Y -530.317,Z 893.034,A 0.000,B 0.000,C 90.000,E1 42.204} C_DIS
LIN {X 0.267,Y -526.835,Z 893.031,A 0.000,B 0.000,C 90.000,E1 41.595} C_DIS
LIN {X -0.200,Y -523.068,Z 893.028,A 0.000,B 0.000,C 90.000,E1 41.067} C_DIS
LIN {X 0.045,Y -519.143,Z 893.025,A 0.000,B 0.000,C 90.000,E1 40.458} C_DIS
LIN {X -0.075,Y -514.921,Z 893.022,A 0.000,B 0.000,C 90.000,E1 39.886} C_DIS
LIN {X 0.050,Y -509.486,Z 893.018,A 0.000,B 0.000,C 90.000,E1 39.152} C_DIS
LIN {X -0.285,Y -503.643,Z 893.014,A 0.000,B 0.000,C 90.000,E1 38.463} C_DIS
LIN {X 0.237,Y -498.404,Z 893.010,A 0.000,B 0.000,C 90.000,E1 37.810} C_DIS
LIN {X 0.167,Y -492.936,Z 893.007,A 0.000,B 0.000,C 90.000,E1 37.237} C_DIS
LIN {X -0.292,Y -486.001,Z 893.003,A 0.000,B 0.000,C 90.000,E1 36.583} C_DIS
LIN {X -0.227,Y -478.722,Z 892.999,A 0.000,B 0.000,C 90.000,E1 35.884} C_DIS
LIN {X -0.107,Y -468.263,Z 892.994,A 0.000,B 0.000,C 90.000,E1 34.945} C_DIS
LIN {X -0.001,Y -455.992,Z 892.988,A 0.000,B 0.000,C 90.000,E1 33.913} C_DIS
LIN {X -0.064,Y -445.097,Z 892.984,A 0.000,B 0.000,C 90.000,E1 33.038} C_DIS
LIN {X -0.008,Y -418.946,Z 892.971,A 0.000,B 0.000,C 90.000,E1 30.846} C_DIS
LIN {X 0.147,Y -402.556,Z 892.963,A 0.000,B 0.000,C 90.000,E1 29.283} C_DIS
LIN {X -0.009,Y -397.310,Z 892.960,A 0.000,B 0.000,C 90.000,E1 28.743} C_DIS
LIN {X -0.107,Y -394.913,Z 892.958,A 0.000,B 0.000,C 90.000,E1 28.437} C_DIS
LIN {X 0.095,Y -393.711,Z 892.957,A 0.000,B 0.000,C 90.000,E1 28.231} C_DIS
LIN {X -0.155,Y -390.698,Z 892.953,A 0.000,B 0.000,C 90.000,E1 27.641} C_DIS
LIN {X 0.049,Y -389.486,Z 892.951,A 0.000,B 0.000,C 90.000,E1 27.078} C_DIS
LIN {X -0.184,Y -388.949,Z 892.947,A 0.000,B 0.000,C 90.000,E1 26.488} C_DIS
LIN {X -0.144,Y -389.082,Z 892.941,A 0.000,B 0.000,C 90.000,E1 25.412} C_DIS
LIN {X -0.115,Y -391.914,Z 892.921,A 0.000,B 0.000,C 90.000,E1 21.844} C_DIS
LIN {X 0.147,Y -394.499,Z 892.908,A 0.000,B 0.000,C 90.000,E1 19.322} C_DIS
LIN {X 0.092,Y -397.342,Z 892.894,A 0.000,B 0.000,C 90.000,E1 16.858} C_DIS
LIN {X -0.148,Y -399.590,Z 892.884,A 0.000,B 0.000,C 90.000,E1 15.134} C_DIS
LIN {X 0.097,Y -403.884,Z 892.867,A 0.000,B 0.000,C 90.000,E1 11.951} C_DIS
LIN {X -0.165,Y -408.113,Z 892.851,A 0.000,B 0.000,C 90.000,E1 9.208} C_DIS
LIN {X -0.027,Y -412.784,Z 892.836,A 0.000,B 0.000,C 90.000,E1 6.429} C_DIS
LIN {X 0.074,Y -416.562,Z 892.824,A 0.000,B 0.000,C 90.000,E1 4.359} C_DIS
LIN {X 0.147,Y -418.649,Z 892.819,A 0.000,B 0.000,C 90.000,E1 3.326} C_DIS
LIN {X 0.033,Y -424.493,Z 892.804,A 0.000,B 0.000,C 90.000,E1 0.630} C_DIS
LIN {X -0.020,Y -429.766,Z 892.791,A 0.000,B 0.000,C 90.000,E1 358.453} C_DIS
LIN {X 0.045,Y -434.939,Z 892.780,A 0.000,B 0.000,C 90.000,E1 356.445} C_DIS
LIN {X 0.176,Y -436.542,Z 892.778,A 0.000,B 0.000,C 90.000,E1 355.931} C_DIS
LIN {X -0.090,Y -438.662,Z 892.775,A 0.000,B 0.000,C 90.000,E1 355.469} C_DIS
LIN {X 0.108,Y -440.165,Z 892.773,A 0.000,B 0.000,C 90.000,E1 355.179} C_DIS
LIN {X -0.088,Y -443.059,Z 892.771,A 0.000,B 0.000,C 90.000,E1 354.837} C_DIS
LIN {X 0.163,Y -443.936,Z 892.771,A 0.000,B 0.000,C 90.000,E1 354.723} C_DIS
LIN {X -0.159,Y -447.926,Z 892.769,A 0.000,B 0.000,C 90.000,E1 354.489} C_DIS
LIN {X -0.179,Y -452.246,Z 892.768,A 0.000,B 0.000,C 90.000,E1 354.261} C_DIS
LIN {X 0.109,Y -465.740,Z 892.765,A 0.000,B 0.000,C 90.000,E1 353.628} C_DIS
LIN {X -0.022,Y -475.965,Z 892.762,A 0.000,B 0.000,C 90.000,E1 353.166} C_DIS
LIN {X -0.058,Y -485.866,Z 892.759,A 0.000,B 0.000,C 90.000,E1 352.648} C_DIS
LIN {X 0.130,Y -498.844,Z 892.755,A 0.000,B 0.000,C 90.000,E1 351.894} C_DIS
LIN {X 0.056,Y -508.476,Z 892.752,A 0.000,B 0.000,C 90.000,E1 351.319} C_DIS
LIN {X 0.126,Y -514.964,Z 892.750,A 0.000,B 0.000,C 90.000,E1 350.905} C_DIS
LIN {X -0.227,Y -524.136,Z 892.746,A 0.000,B 0.000,C 90.000,E1 350.330} C_DIS
LIN {X 0.073,Y -531.715,Z 892.743,A 0.000,B 0.000,C 90.000,E1 349.746} C_DIS
LIN {X 0.025,Y -538.916,Z 892.740,A 0.000,B 0.000,C 90.000,E1 349.162} C_DIS
LIN {X -0.207,Y -545.934,Z 892.736,A 0.000,B 0.000,C 90.000,E1 348.578} C_DIS
LIN {X -0.115,Y -552.628,Z 892.733,A 0.000,B 0.000,C 90.000,E1 347.937} C_DIS
LIN {X 0.257,Y -559.074,Z 892.729,A 0.000,B 0.000,C 90.000,E1 347.229} C_DIS
LIN {X 0.242,Y -562.799,Z 892.727,A 0.000,B 0.000,C 90.000,E1 346.825} C_DIS
LIN {X 0.315,Y -569.837,Z 892.722,A 0.000,B 0.000,C 90.000,E1 345.992} C_DIS
LIN {X -0.314,Y -573.116,Z 892.720,A 0.000,B 0.000,C 90.000,E1 345.644} C_DIS
LIN {X -0.132,Y -579.303,Z 892.716,A 0.000,B 0.000,C 90.000,E1 344.810} C_DIS
LIN {X 0.207,Y -584.206,Z 892.712,A 0.000,B 0.000,C 90.000,E1 344.102} C_DIS
LIN {X 0.026,Y -588.699,Z 892.708,A 0.000,B 0.000,C 90.000,E1 343.449} C_DIS
LIN {X 0.246,Y -595.305,Z 892.702,A 0.000,B 0.000,C 90.000,E1 342.362} C_DIS
LIN {X 0.047,Y -600.592,Z 892.697,A 0.000,B 0.000,C 90.000,E1 341.456} C_DIS
LIN {X -0.092,Y -605.577,Z 892.692,A 0.000,B 0.000,C 90.000,E1 340.550} C_DIS
LIN {X -0.210,Y -610.991,Z 892.686,A 0.000,B 0.000,C 90.000,E1 339.518} C_DIS
LIN {X -0.037,Y -616.099,Z 892.680,A 0.000,B 0.000,C 90.000,E1 338.465} C_DIS
LIN {X -0.031,Y -621.469,Z 892.674,A 0.000,B 0.000,C 90.000,E1 337.305} C_DIS
LIN {X -0.298,Y -625.951,Z 892.668,A 0.000,B 0.000,C 90.000,E1 336.305} C_DIS
LIN {X 0.328,Y -630.117,Z 892.663,A 0.000,B 0.000,C 90.000,E1 335.229} C_DIS
LIN {X -0.359,Y -634.892,Z 892.656,A 0.000,B 0.000,C 90.000,E1 334.024} C_DIS
LIN {X -0.226,Y -637.613,Z 892.651,A 0.000,B 0.000,C 90.000,E1 333.256} C_DIS
LIN {X 0.054,Y -641.801,Z 892.644,A 0.000,B 0.000,C 90.000,E1 331.975} C_DIS
LIN {X 0.143,Y -645.542,Z 892.637,A 0.000,B 0.000,C 90.000,E1 330.717} C_DIS
LIN {X -0.107,Y -648.413,Z 892.632,A 0.000,B 0.000,C 90.000,E1 329.744} C_DIS
LIN {X 0.002,Y -651.137,Z 892.626,A 0.000,B 0.000,C 90.000,E1 328.742} C_DIS
LIN {X 0.055,Y -653.073,Z 892.622,A 0.000,B 0.000,C 90.000,E1 327.995} C_DIS
LIN {X 0.130,Y -654.830,Z 892.618,A 0.000,B 0.000,C 90.000,E1 327.248} C_DIS
LIN {X -0.231,Y -656.966,Z 892.613,A 0.000,B 0.000,C 90.000,E1 326.294} C_DIS
LIN {X -0.104,Y -659.225,Z 892.606,A 0.000,B 0.000,C 90.000,E1 325.055} C_DIS
LIN {X -0.136,Y -660.400,Z 892.602,A 0.000,B 0.000,C 90.000,E1 324.322} C_DIS
LIN {X -0.054,Y -661.795,Z 892.596,A 0.000,B 0.000,C 90.000,E1 323.336} C_DIS
LIN {X -0.436,Y -663.402,Z 892.588,A 0.000,B 0.000,C 90.000,E1 321.904} C_DIS
LIN {X 0.058,Y -664.670,Z 892.581,A 0.000,B 0.000,C 90.000,E1 320.642} C_DIS
LIN {X -0.362,Y -665.906,Z 892.575,A 0.000,B 0.000,C 90.000,E1 319.461} C_DIS
LIN {X 0.156,Y -667.647,Z 892.565,A 0.000,B 0.000,C 90.000,E1 317.715} C_DIS
LIN {X -0.279,Y -669.286,Z 892.557,A 0.000,B 0.000,C 90.000,E1 316.296} C_DIS
LIN {X -0.216,Y -670.691,Z 892.549,A 0.000,B 0.000,C 90.000,E1 314.838} C_DIS
LIN {X 0.414,Y -672.793,Z 892.537,A 0.000,B 0.000,C 90.000,E1 312.609} C_DIS
LIN {X 0.051,Y -673.951,Z 892.530,A 0.000,B 0.000,C 90.000,E1 311.434} C_DIS
LIN {X 0.320,Y -675.362,Z 892.521,A 0.000,B 0.000,C 90.000,E1 309.725} C_DIS
LIN {X 0.083,Y -676.576,Z 892.513,A 0.000,B 0.000,C 90.000,E1 308.302} C_DIS
LIN {X 0.376,Y -677.420,Z 892.506,A 0.000,B 0.000,C 90.000,E1 307.076} C_DIS
LIN {X -0.111,Y -678.422,Z 892.498,A 0.000,B 0.000,C 90.000,E1 305.678} C_DIS
LIN {X -0.020,Y -679.346,Z 892.489,A 0.000,B 0.000,C 90.000,E1 303.992} C_DIS
LIN {X -0.110,Y -680.541,Z 892.478,A 0.000,B 0.000,C 90.000,E1 302.084} C_DIS
LIN {X 0.406,Y -682.019,Z 892.468,A 0.000,B 0.000,C 90.000,E1 300.129} C_DIS
LIN {X 0.093,Y -684.444,Z 892.454,A 0.000,B 0.000,C 90.000,E1 297.769} C_DIS
LIN {X 0.309,Y -686.734,Z 892.444,A 0.000,B 0.000,C 90.000,E1 295.848} C_DIS
LIN {X -0.107,Y -688.193,Z 892.437,A 0.000,B 0.000,C 90.000,E1 294.695} C_DIS
LIN {X -0.164,Y -689.274,Z 892.431,A 0.000,B 0.000,C 90.000,E1 293.515} C_DIS
LIN {X 0.248,Y -689.006,Z 892.427,A 0.000,B 0.000,C 90.000,E1 292.770} C_DIS
LIN {X -0.203,Y -687.899,Z 892.424,A 0.000,B 0.000,C 90.000,E1 292.333} C_DIS
LIN {X 0.018,Y -687.122,Z 892.423,A 0.000,B 0.000,C 90.000,E1 292.078} C_DIS
LIN {X -0.130,Y -686.354,Z 892.422,A 0.000,B 0.000,C 90.000,E1 291.972} C_DIS
LIN {X 0.190,Y -683.085,Z 892.420,A 0.000,B 0.000,C 90.000,E1 291.589} C_DIS
LIN {X 0.291,Y -681.957,Z 892.419,A 0.000,B 0.000,C 90.000,E1 291.461} C_DIS
LIN {X 0.143,Y -680.587,Z 892.419,A 0.000,B 0.000,C 90.000,E1 291.354} C_DIS
LIN {X -0.298,Y -678.527,Z 892.418,A 0.000,B 0.000,C 90.000,E1 291.280} C_DIS
LIN {X -0.219,Y -668.620,Z 892.416,A 0.000,B 0.000,C 90.000,E1 290.918} C_DIS
LIN {X -0.155,Y -664.440,Z 892.415,A 0.000,B 0.000,C 90.000,E1 290.791} C_DIS
LIN {X 0.342,Y -661.132,Z 892.415,A 0.000,B 0.000,C 90.000,E1 290.610} C_DIS
LIN {X 0.164,Y -658.249,Z 892.414,A 0.000,B 0.000,C 90.000,E1 290.482} C_DIS
LIN {X 0.107,Y -658.190,Z 892.414,A 0.000,B 0.000,C 90.000,E1 290.482} C_DIS
LIN {X 0.058,Y -657.488,Z 892.413,A 0.000,B 0.000,C 90.000,E1 290.375} C_DIS
LIN {X 0.014,Y -657.474,Z 892.413,A 0.000,B 0.000,C 90.000,E1 290.375} C_DIS
LIN {X -0.013,Y -657.476,Z 892.412,A 0.000,B 0.000,C 90.000,E1 290.174} C_DIS
LIN {X -0.135,Y -658.126,Z 892.411,A 0.000,B 0.000,C 90.000,E1 289.939} C_DIS
LIN {X -0.034,Y -658.909,Z 892.409,A 0.000,B 0.000,C 90.000,E1 289.685} C_DIS
LIN {X -0.160,Y -662.379,Z 892.405,A 0.000,B 0.000,C 90.000,E1 288.960} C_DIS
LIN {X -0.247,Y -666.255,Z 892.401,A 0.000,B 0.000,C 90.000,E1 288.236} C_DIS
LIN {X -0.218,Y -668.755,Z 892.399,A 0.000,B 0.000,C 90.000,E1 287.747} C_DIS
LIN {X 0.192,Y -672.136,Z 892.394,A 0.000,B 0.000,C 90.000,E1 286.985} C_DIS
LIN {X 0.254,Y -674.113,Z 892.392,A 0.000,B 0.000,C 90.000,E1 286.496} C_DIS
LIN {X 0.084,Y -676.518,Z 892.388,A 0.000,B 0.000,C 90.000,E1 285.788} C_DIS
LIN {X 0.117,Y -678.364,Z 892.384,A 0.000,B 0.000,C 90.000,E1 285.064} C_DIS
LIN {X -0.012,Y -679.922,Z 892.380,A 0.000,B 0.000,C 90.000,E1 284.356} C_DIS
LIN {X -0.124,Y -681.243,Z 892.376,A 0.000,B 0.000,C 90.000,E1 283.647} C_DIS
LIN {X -0.259,Y -682.594,Z 892.370,A 0.000,B 0.000,C 90.000,E1 282.703} C_DIS
LIN {X 0.201,Y -683.079,Z 892.368,A 0.000,B 0.000,C 90.000,E1 282.187} C_DIS
LIN {X 0.116,Y -683.478,Z 892.364,A 0.000,B 0.000,C 90.000,E1 281.478} C_DIS
LIN {X 0.086,Y -683.550,Z 892.363,A 0.000,B 0.000,C 90.000,E1 281.243} C_DIS
LIN {X -0.133,Y -683.146,Z 892.359,A 0.000,B 0.000,C 90.000,E1 280.546} C_DIS
LIN {X -0.197,Y -682.641,Z 892.356,A 0.000,B 0.000,C 90.000,E1 280.074} C_DIS
LIN {X 0.287,Y -681.809,Z 892.353,A 0.000,B 0.000,C 90.000,E1 279.557} C_DIS
LIN {X 0.098,Y -680.619,Z 892.351,A 0.000,B 0.000,C 90.000,E1 279.095} C_DIS
LIN {X 0.008,Y -679.113,Z 892.348,A 0.000,B 0.000,C 90.000,E1 278.624} C_DIS
LIN {X -0.347,Y -676.391,Z 892.344,A 0.000,B 0.000,C 90.000,E1 277.936} C_DIS
LIN {X 0.195,Y -674.192,Z 892.341,A 0.000,B 0.000,C 90.000,E1 277.409} C_DIS
LIN {X -0.117,Y -671.098,Z 892.338,A 0.000,B 0.000,C 90.000,E1 276.834} C_DIS
LIN {X 0.211,Y -667.577,Z 892.335,A 0.000,B 0.000,C 90.000,E1 276.201} C_DIS
LIN {X 0.023,Y -665.345,Z 892.333,A 0.000,B 0.000,C 90.000,E1 275.853} C_DIS
LIN {X 0.301,Y -660.974,Z 892.329,A 0.000,B 0.000,C 90.000,E1 275.220} C_DIS
LIN {X -0.019,Y -657.000,Z 892.326,A 0.000,B 0.000,C 90.000,E1 274.759} C_DIS
LIN {X 0.135,Y -651.341,Z 892.323,A 0.000,B 0.000,C 90.000,E1 274.131} C_DIS
LIN {X -0.151,Y -646.444,Z 892.320,A 0.000,B 0.000,C 90.000,E1 273.669} C_DIS
LIN {X -0.273,Y -639.874,Z 892.317,A 0.000,B 0.000,C 90.000,E1 273.094} C_DIS
LIN {X -0.216,Y -634.370,Z 892.315,A 0.000,B 0.000,C 90.000,E1 272.636} C_DIS
LIN {X 0.042,Y -630.112,Z 892.313,A 0.000,B 0.000,C 90.000,E1 272.293} C_DIS
LIN {X 0.092,Y -624.331,Z 892.311,A 0.000,B 0.000,C 90.000,E1 271.892} C_DIS
LIN {X 0.003,Y -616.509,Z 892.308,A 0.000,B 0.000,C 90.000,E1 271.432} C_DIS
LIN {X -0.081,Y -609.861,Z 892.306,A 0.000,B 0.000,C 90.000,E1 271.088} C_DIS
LIN {X 0.262,Y -603.275,Z 892.304,A 0.000,B 0.000,C 90.000,E1 270.745} C_DIS
LIN {X 0.270,Y -597.999,Z 892.303,A 0.000,B 0.000,C 90.000,E1 270.516} C_DIS
LIN {X -0.140,Y -590.870,Z 892.302,A 0.000,B 0.000,C 90.000,E1 270.286} C_DIS
LIN {X -0.211,Y -583.539,Z 892.300,A 0.000,B 0.000,C 90.000,E1 270.057} C_DIS
LIN {X 0.020,Y -577.882,Z 892.299,A 0.000,B 0.000,C 90.000,E1 269.885} C_DIS
LIN {X -0.121,Y -571.552,Z 892.299,A 0.000,B 0.000,C 90.000,E1 269.771} C_DIS
LIN {X 0.111,Y -565.004,Z 892.298,A 0.000,B 0.000,C 90.000,E1 269.656} C_DIS
LIN {X 0.212,Y -552.449,Z 892.298,A 0.000,B 0.000,C 90.000,E1 269.542} C_DIS
LIN {X -0.155,Y -549.511,Z 892.297,A 0.000,B 0.000,C 90.000,E1 269.484} C_DIS
LIN {X -0.190,Y -549.436,Z 892.297,A 0.000,B 0.000,C 90.000,E1 269.484} C_DIS
LIN {X 0.054,Y -546.875,Z 892.295,A 0.000,B 0.000,C 90.000,E1 269.141} C_DIS
LIN {X -0.024,Y -545.256,Z 892.293,A 0.000,B 0.000,C 90.000,E1 268.797} C_DIS
LIN {X 0.178,Y -544.356,Z 892.291,A 0.000,B 0.000,C 90.000,E1 268.282} C_DIS
LIN {X -0.108,Y -542.220,Z 892.280,A 0.000,B 0.000,C 90.000,E1 266.331} C_DIS
LIN {X 0.154,Y -540.654,Z 892.267,A 0.000,B 0.000,C 90.000,E1 264.033} C_DIS
LIN {X -0.182,Y -539.896,Z 892.261,A 0.000,B 0.000,C 90.000,E1 262.932} C_DIS
LIN {X -0.059,Y -538.897,Z 892.254,A 0.000,B 0.000,C 90.000,E1 261.781} C_DIS
LIN {X 0.182,Y -537.485,Z 892.246,A 0.000,B 0.000,C 90.000,E1 260.330} C_DIS
LIN {X 0.085,Y -535.431,Z 892.235,A 0.000,B 0.000,C 90.000,E1 258.342} C_DIS
LIN {X -0.215,Y -534.199,Z 892.229,A 0.000,B 0.000,C 90.000,E1 257.229} C_DIS
LIN {X -0.019,Y -532.711,Z 892.223,A 0.000,B 0.000,C 90.000,E1 256.061} C_DIS
LIN {X 0.141,Y -530.180,Z 892.211,A 0.000,B 0.000,C 90.000,E1 254.031} C_DIS
LIN {X 0.059,Y -528.429,Z 892.203,A 0.000,B 0.000,C 90.000,E1 252.598} C_DIS
LIN {X -0.071,Y -527.051,Z 892.197,A 0.000,B 0.000,C 90.000,E1 251.456} C_DIS
LIN {X 0.108,Y -524.869,Z 892.187,A 0.000,B 0.000,C 90.000,E1 249.699} C_DIS
LIN {X -0.073,Y -522.489,Z 892.178,A 0.000,B 0.000,C 90.000,E1 247.975} C_DIS
LIN {X -0.104,Y -519.958,Z 892.168,A 0.000,B 0.000,C 90.000,E1 246.230} C_DIS
LIN {X 0.021,Y -517.258,Z 892.158,A 0.000,B 0.000,C 90.000,E1 244.460} C_DIS
LIN {X -0.055,Y -515.892,Z 892.153,A 0.000,B 0.000,C 90.000,E1 243.589} C_DIS
LIN {X 0.080,Y -513.420,Z 892.145,A 0.000,B 0.000,C 90.000,E1 242.103} C_DIS
LIN {X 0.075,Y -511.354,Z 892.139,A 0.000,B 0.000,C 90.000,E1 240.923} C_DIS
LIN {X 0.004,Y -508.235,Z 892.129,A 0.000,B 0.000,C 90.000,E1 239.154} C_DIS
LIN {X -0.043,Y -505.097,Z 892.119,A 0.000,B 0.000,C 90.000,E1 237.375} C_DIS
LIN {X 0.077,Y -502.674,Z 892.112,A 0.000,B 0.000,C 90.000,E1 236.167} C_DIS
LIN {X 0.140,Y -500.684,Z 892.107,A 0.000,B 0.000,C 90.000,E1 235.261} C_DIS
LIN {X -0.206,Y -496.485,Z 892.097,A 0.000,B 0.000,C 90.000,E1 233.497} C_DIS
LIN {X -0.041,Y -492.426,Z 892.087,A 0.000,B 0.000,C 90.000,E1 231.662} C_DIS
LIN {X -0.130,Y -487.632,Z 892.075,A 0.000,B 0.000,C 90.000,E1 229.542} C_DIS
LIN {X -0.042,Y -484.182,Z 892.067,A 0.000,B 0.000,C 90.000,E1 228.000} C_DIS
LIN {X -0.021,Y -480.713,Z 892.058,A 0.000,B 0.000,C 90.000,E1 226.458} C_DIS
LIN {X -0.200,Y -477.969,Z 892.051,A 0.000,B 0.000,C 90.000,E1 225.243} C_DIS
LIN {X 0.254,Y -475.130,Z 892.044,A 0.000,B 0.000,C 90.000,E1 223.947} C_DIS
LIN {X -0.244,Y -471.626,Z 892.036,A 0.000,B 0.000,C 90.000,E1 222.447} C_DIS
LIN {X -0.103,Y -468.115,Z 892.027,A 0.000,B 0.000,C 90.000,E1 220.862} C_DIS
LIN {X 0.022,Y -464.050,Z 892.016,A 0.000,B 0.000,C 90.000,E1 218.955} C_DIS
LIN {X 0.049,Y -461.420,Z 892.009,A 0.000,B 0.000,C 90.000,E1 217.684} C_DIS
LIN {X -0.203,Y -457.318,Z 891.999,A 0.000,B 0.000,C 90.000,E1 215.804} C_DIS
LIN {X -0.073,Y -453.294,Z 891.988,A 0.000,B 0.000,C 90.000,E1 213.865} C_DIS
LIN {X 0.112,Y -447.730,Z 891.974,A 0.000,B 0.000,C 90.000,E1 211.258} C_DIS
LIN {X -0.034,Y -442.750,Z 891.961,A 0.000,B 0.000,C 90.000,E1 208.999} C_DIS
LIN {X 0.209,Y -438.418,Z 891.950,A 0.000,B 0.000,C 90.000,E1 207.001} C_DIS
LIN {X -0.018,Y -433.405,Z 891.937,A 0.000,B 0.000,C 90.000,E1 204.719} C_DIS
LIN {X -0.177,Y -429.798,Z 891.928,A 0.000,B 0.000,C 90.000,E1 203.078} C_DIS
LIN {X 0.015,Y -425.626,Z 891.917,A 0.000,B 0.000,C 90.000,E1 201.046} C_DIS
LIN {X -0.224,Y -422.129,Z 891.908,A 0.000,B 0.000,C 90.000,E1 199.396} C_DIS
LIN {X 0.026,Y -418.052,Z 891.896,A 0.000,B 0.000,C 90.000,E1 197.330} C_DIS
LIN {X 0.171,Y -414.518,Z 891.887,A 0.000,B 0.000,C 90.000,E1 195.607} C_DIS
LIN {X -0.126,Y -410.488,Z 891.875,A 0.000,B 0.000,C 90.000,E1 193.592} C_DIS
LIN {X 0.166,Y -407.235,Z 891.866,A 0.000,B 0.000,C 90.000,E1 191.827} C_DIS
LIN {X -0.177,Y -404.516,Z 891.858,A 0.000,B 0.000,C 90.000,E1 190.489} C_DIS
LIN {X -0.161,Y -400.947,Z 891.849,A 0.000,B 0.000,C 90.000,E1 188.746} C_DIS
LIN {X 0.098,Y -396.807,Z 891.837,A 0.000,B 0.000,C 90.000,E1 186.606} C_DIS
LIN {X 0.073,Y -391.748,Z 891.821,A 0.000,B 0.000,C 90.000,E1 183.784} C_DIS
LIN {X -0.011,Y -388.388,Z 891.809,A 0.000,B 0.000,C 90.000,E1 181.661} C_DIS
LIN {X -0.094,Y -385.725,Z 891.799,A 0.000,B 0.000,C 90.000,E1 179.885} C_DIS
LIN {X 0.052,Y -382.429,Z 891.787,A 0.000,B 0.000,C 90.000,E1 177.707} C_DIS
LIN {X -0.082,Y -376.747,Z 891.765,A 0.000,B 0.000,C 90.000,E1 173.742} C_DIS
LIN {X -0.184,Y -375.527,Z 891.757,A 0.000,B 0.000,C 90.000,E1 172.299} C_DIS
LIN {X -0.114,Y -375.145,Z 891.752,A 0.000,B 0.000,C 90.000,E1 171.376} C_DIS
LIN {X 0.022,Y -375.382,Z 891.748,A 0.000,B 0.000,C 90.000,E1 170.557} C_DIS
LIN {X 0.085,Y -376.160,Z 891.743,A 0.000,B 0.000,C 90.000,E1 169.634} C_DIS
LIN {X -0.043,Y -377.197,Z 891.740,A 0.000,B 0.000,C 90.000,E1 169.106} C_DIS
LIN {X -0.061,Y -377.437,Z 891.738,A 0.000,B 0.000,C 90.000,E1 168.926} C_DIS
LIN {X 0.191,Y -378.997,Z 891.735,A 0.000,B 0.000,C 90.000,E1 168.342} C_DIS
LIN {X -0.129,Y -379.742,Z 891.734,A 0.000,B 0.000,C 90.000,E1 168.117} C_DIS
LIN {X -0.006,Y -382.150,Z 891.731,A 0.000,B 0.000,C 90.000,E1 167.645} C_DIS
LIN {X 0.195,Y -385.058,Z 891.729,A 0.000,B 0.000,C 90.000,E1 167.173} C_DIS
LIN {X 0.194,Y -386.523,Z 891.728,A 0.000,B 0.000,C 90.000,E1 166.992} C_DIS
LIN {X -0.080,Y -391.525,Z 891.725,A 0.000,B 0.000,C 90.000,E1 166.520} C_DIS
LIN {X -0.162,Y -395.728,Z 891.723,A 0.000,B 0.000,C 90.000,E1 166.228} C_DIS
LIN {X 0.194,Y -407.403,Z 891.719,A 0.000,B 0.000,C 90.000,E1 165.463} C_DIS
LIN {X 0.167,Y -412.626,Z 891.718,A 0.000,B 0.000,C 90.000,E1 165.172} C_DIS
LIN {X -0.093,Y -419.201,Z 891.716,A 0.000,B 0.000,C 90.000,E1 164.810} C_DIS
LIN {X -0.047,Y -428.671,Z 891.712,A 0.000,B 0.000,C 90.000,E1 164.157} C_DIS
LIN {X 0.023,Y -435.119,Z 891.709,A 0.000,B 0.000,C 90.000,E1 163.685} C_DIS
LIN {X -0.081,Y -444.115,Z 891.705,A 0.000,B 0.000,C 90.000,E1 162.960} C_DIS
LIN {X -0.049,Y -451.643,Z 891.702,A 0.000,B 0.000,C 90.000,E1 162.308} C_DIS
LIN {X -0.098,Y -458.866,Z 891.698,A 0.000,B 0.000,C 90.000,E1 161.638} C_DIS
LIN {X -0.009,Y -467.498,Z 891.693,A 0.000,B 0.000,C 90.000,E1 160.786} C_DIS
LIN {X -0.071,Y -471.514,Z 891.691,A 0.000,B 0.000,C 90.000,E1 160.369} C_DIS
LIN {X 0.229,Y -479.663,Z 891.686,A 0.000,B 0.000,C 90.000,E1 159.444} C_DIS
LIN {X -0.033,Y -483.517,Z 891.684,A 0.000,B 0.000,C 90.000,E1 159.028} C_DIS
LIN {X 0.033,Y -493.320,Z 891.677,A 0.000,B 0.000,C 90.000,E1 157.794} C_DIS
LIN {X -0.222,Y -502.259,Z 891.670,A 0.000,B 0.000,C 90.000,E1 156.613} C_DIS
LIN {X -0.051,Y -507.638,Z 891.666,A 0.000,B 0.000,C 90.000,E1 155.845} C_DIS
LIN {X -0.214,Y -513.959,Z 891.661,A 0.000,B 0.000,C 90.000,E1 154.973} C_DIS
LIN {X -0.089,Y -519.863,Z 891.656,A 0.000,B 0.000,C 90.000,E1 154.076} C_DIS
LIN {X 0.028,Y -524.908,Z 891.652,A 0.000,B 0.000,C 90.000,E1 153.332} C_DIS
LIN {X 0.222,Y -532.443,Z 891.646,A 0.000,B 0.000,C 90.000,E1 152.153} C_DIS
LIN {X 0.112,Y -535.922,Z 891.642,A 0.000,B 0.000,C 90.000,E1 151.591} C_DIS
LIN {X -0.124,Y -545.020,Z 891.634,A 0.000,B 0.000,C 90.000,E1 150.049} C_DIS
LIN {X -0.135,Y -549.566,Z 891.629,A 0.000,B 0.000,C 90.000,E1 149.203} C_DIS
LIN {X 0.012,Y -553.429,Z 891.625,A 0.000,B 0.000,C 90.000,E1 148.486} C_DIS
LIN {X -0.271,Y -563.040,Z 891.615,A 0.000,B 0.000,C 90.000,E1 146.707} C_DIS
LIN {X -0.268,Y -569.153,Z 891.608,A 0.000,B 0.000,C 90.000,E1 145.468} C_DIS
LIN {X 0.213,Y -576.917,Z 891.599,A 0.000,B 0.000,C 90.000,E1 143.783} C_DIS
LIN {X -0.122,Y -580.640,Z 891.594,A 0.000,B 0.000,C 90.000,E1 143.004} C_DIS
LIN {X 0.023,Y -586.084,Z 891.588,A 0.000,B 0.000,C 90.000,E1 141.778} C_DIS
LIN {X -0.011,Y -592.568,Z 891.580,A 0.000,B 0.000,C 90.000,E1 140.312} C_DIS
LIN {X -0.289,Y -595.997,Z 891.575,A 0.000,B 0.000,C 90.000,E1 139.542} C_DIS
LIN {X 0.330,Y -601.778,Z 891.568,A 0.000,B 0.000,C 90.000,E1 138.162} C_DIS
LIN {X -0.372,Y -605.853,Z 891.563,A 0.000,B 0.000,C 90.000,E1 137.310} C_DIS
LIN {X -0.175,Y -609.940,Z 891.558,A 0.000,B 0.000,C 90.000,E1 136.377} C_DIS
LIN {X 0.079,Y -617.013,Z 891.549,A 0.000,B 0.000,C 90.000,E1 134.798} C_DIS
LIN {X -0.106,Y -621.487,Z 891.543,A 0.000,B 0.000,C 90.000,E1 133.785} C_DIS
LIN {X -0.363,Y -627.058,Z 891.536,A 0.000,B 0.000,C 90.000,E1 132.528} C_DIS
LIN {X -0.179,Y -633.410,Z 891.528,A 0.000,B 0.000,C 90.000,E1 130.987} C_DIS
LIN {X -0.075,Y -637.598,Z 891.522,A 0.000,B 0.000,C 90.000,E1 129.967} C_DIS
LIN {X 0.105,Y -640.592,Z 891.518,A 0.000,B 0.000,C 90.000,E1 129.197} C_DIS
LIN {X -0.174,Y -645.382,Z 891.511,A 0.000,B 0.000,C 90.000,E1 127.971} C_DIS
LIN {X 0.017,Y -650.133,Z 891.504,A 0.000,B 0.000,C 90.000,E1 126.710} C_DIS
LIN {X 0.031,Y -654.624,Z 891.497,A 0.000,B 0.000,C 90.000,E1 125.471} C_DIS
LIN {X 0.044,Y -658.024,Z 891.492,A 0.000,B 0.000,C 90.000,E1 124.485} C_DIS
LIN {X 0.205,Y -662.010,Z 891.485,A 0.000,B 0.000,C 90.000,E1 123.245} C_DIS
LIN {X 0.247,Y -663.440,Z 891.482,A 0.000,B 0.000,C 90.000,E1 122.752} C_DIS
LIN {X 0.135,Y -666.734,Z 891.475,A 0.000,B 0.000,C 90.000,E1 121.544} C_DIS
LIN {X 0.346,Y -668.377,Z 891.471,A 0.000,B 0.000,C 90.000,E1 120.797} C_DIS
LIN {X -0.030,Y -670.690,Z 891.465,A 0.000,B 0.000,C 90.000,E1 119.617} C_DIS
LIN {X 0.377,Y -672.229,Z 891.459,A 0.000,B 0.000,C 90.000,E1 118.615} C_DIS
LIN {X -0.079,Y -674.348,Z 891.451,A 0.000,B 0.000,C 90.000,E1 117.206} C_DIS
LIN {X 0.047,Y -675.389,Z 891.446,A 0.000,B 0.000,C 90.000,E1 116.232} C_DIS
LIN {X -0.116,Y -676.080,Z 891.440,A 0.000,B 0.000,C 90.000,E1 115.283} C_DIS
LIN {X -0.174,Y -676.313,Z 891.436,A 0.000,B 0.000,C 90.000,E1 114.567} C_DIS
LIN {X -0.083,Y -676.293,Z 891.434,A 0.000,B 0.000,C 90.000,E1 114.079} C_DIS
LIN {X 0.014,Y -675.994,Z 891.431,A 0.000,B 0.000,C 90.000,E1 113.590} C_DIS
LIN {X 0.197,Y -675.761,Z 891.430,A 0.000,B 0.000,C 90.000,E1 113.334} C_DIS
LIN {X -0.326,Y -674.616,Z 891.427,A 0.000,B 0.000,C 90.000,E1 112.898} C_DIS
LIN {X -0.149,Y -673.692,Z 891.426,A 0.000,B 0.000,C 90.000,E1 112.642} C_DIS
LIN {X 0.025,Y -672.111,Z 891.424,A 0.000,B 0.000,C 90.000,E1 112.386} C_DIS
LIN {X -0.063,Y -670.317,Z 891.423,A 0.000,B 0.000,C 90.000,E1 112.153} C_DIS
LIN {X 0.017,Y -669.283,Z 891.422,A 0.000,B 0.000,C 90.000,E1 112.025} C_DIS
LIN {X 0.097,Y -667.694,Z 891.422,A 0.000,B 0.000,C 90.000,E1 111.897} C_DIS
LIN {X 0.114,Y -665.704,Z 891.421,A 0.000,B 0.000,C 90.000,E1 111.791} C_DIS
LIN {X -0.125,Y -662.486,Z 891.420,A 0.000,B 0.000,C 90.000,E1 111.589} C_DIS
LIN {X 0.205,Y -660.487,Z 891.419,A 0.000,B 0.000,C 90.000,E1 111.461} C_DIS
LIN {X -0.164,Y -656.053,Z 891.419,A 0.000,B 0.000,C 90.000,E1 111.334} C_DIS
LIN {X -0.247,Y -654.084,Z 891.418,A 0.000,B 0.000,C 90.000,E1 111.280} C_DIS
LIN {X 0.252,Y -645.643,Z 891.417,A 0.000,B 0.000,C 90.000,E1 111.046} C_DIS
LIN {X -0.100,Y -631.436,Z 891.416,A 0.000,B 0.000,C 90.000,E1 110.791} C_DIS
LIN {X 0.260,Y -618.164,Z 891.414,A 0.000,B 0.000,C 90.000,E1 110.429} C_DIS
LIN {X 0.237,Y -612.510,Z 891.413,A 0.000,B 0.000,C 90.000,E1 110.248} C_DIS
LIN {X -0.320,Y -603.993,Z 891.411,A 0.000,B 0.000,C 90.000,E1 109.939} C_DIS
LIN {X 0.106,Y -595.069,Z 891.408,A 0.000,B 0.000,C 90.000,E1 109.450} C_DIS
LIN {X 0.102,Y -587.312,Z 891.406,A 0.000,B 0.000,C 90.000,E1 109.033} C_DIS
LIN {X -0.182,Y -580.645,Z 891.404,A 0.000,B 0.000,C 90.000,E1 108.725} C_DIS
LIN {X -0.142,Y -571.543,Z 891.402,A 0.000,B 0.000,C 90.000,E1 108.362} C_DIS
LIN {X -0.171,Y -564.362,Z 891.401,A 0.000,B 0.000,C 90.000,E1 108.109} C_DIS
LIN {X -0.162,Y -561.961,Z 891.400,A 0.000,B 0.000,C 90.000,E1 108.000} C_DIS
LIN {X -0.286,Y -558.469,Z 891.399,A 0.000,B 0.000,C 90.000,E1 107.819} C_DIS
LIN {X 0.191,Y -558.417,Z 891.399,A 0.000,B 0.000,C 90.000,E1 107.764} C_DIS
LIN {X -0.212,Y -557.030,Z 891.398,A 0.000,B 0.000,C 90.000,E1 107.583} C_DIS
LIN {X 0.077,Y -556.470,Z 891.396,A 0.000,B 0.000,C 90.000,E1 107.275} C_DIS
LIN {X -0.178,Y -556.258,Z 891.394,A 0.000,B 0.000,C 90.000,E1 106.985} C_DIS
LIN {X -0.307,Y -556.229,Z 891.391,A 0.000,B 0.000,C 90.000,E1 106.441} C_DIS
LIN {X 0.084,Y -557.034,Z 891.379,A 0.000,B 0.000,C 90.000,E1 104.175} C_DIS
LIN {X 0.238,Y -558.390,Z 891.365,A 0.000,B 0.000,C 90.000,E1 101.658} C_DIS
LIN {X 0.146,Y -559.779,Z 891.354,A 0.000,B 0.000,C 90.000,E1 99.726} C_DIS
LIN {X 0.149,Y -560.803,Z 891.346,A 0.000,B 0.000,C 90.000,E1 98.341} C_DIS
LIN {X -0.083,Y -561.955,Z 891.336,A 0.000,B 0.000,C 90.000,E1 96.429} C_DIS
LIN {X 0.043,Y -562.843,Z 891.327,A 0.000,B 0.000,C 90.000,E1 94.759} C_DIS
LIN {X -0.095,Y -563.347,Z 891.320,A 0.000,B 0.000,C 90.000,E1 93.669} C_DIS
LIN {X 0.114,Y -564.066,Z 891.310,A 0.000,B 0.000,C 90.000,E1 91.718} C_DIS
LIN {X -0.021,Y -564.434,Z 891.304,A 0.000,B 0.000,C 90.000,E1 90.630} C_DIS
LIN {X -0.038,Y -564.732,Z 891.296,A 0.000,B 0.000,C 90.000,E1 89.255} C_DIS
LIN {X 0.074,Y -565.066,Z 891.287,A 0.000,B 0.000,C 90.000,E1 87.593} C_DIS
LIN {X -0.234,Y -565.358,Z 891.276,A 0.000,B 0.000,C 90.000,E1 85.698} C_DIS
LIN {X 0.168,Y -565.762,Z 891.264,A 0.000,B 0.000,C 90.000,E1 83.457} C_DIS
LIN {X -0.121,Y -566.154,Z 891.255,A 0.000,B 0.000,C 90.000,E1 81.837} C_DIS
LIN {X 0.082,Y -566.554,Z 891.247,A 0.000,B 0.000,C 90.000,E1 80.443} C_DIS
LIN {X -0.266,Y -567.079,Z 891.239,A 0.000,B 0.000,C 90.000,E1 79.106} C_DIS
LIN {X 0.059,Y -567.754,Z 891.232,A 0.000,B 0.000,C 90.000,E1 77.701} C_DIS
LIN {X 0.014,Y -568.515,Z 891.223,A 0.000,B 0.000,C 90.000,E1 76.061} C_DIS
LIN {X -0.064,Y -569.142,Z 891.215,A 0.000,B 0.000,C 90.000,E1 74.700} C_DIS
LIN {X 0.023,Y -569.686,Z 891.207,A 0.000,B 0.000,C 90.000,E1 73.323} C_DIS
LIN {X 0.088,Y -570.241,Z 891.197,A 0.000,B 0.000,C 90.000,E1 71.402} C_DIS
LIN {X -0.163,Y -570.532,Z 891.189,A 0.000,B 0.000,C 90.000,E1 70.061} C_DIS
LIN {X -0.236,Y -570.773,Z 891.179,A 0.000,B 0.000,C 90.000,E1 68.156} C_DIS
LIN {X -0.088,Y -570.917,Z 891.168,A 0.000,B 0.000,C 90.000,E1 66.230} C_DIS
LIN {X -0.061,Y -570.910,Z 891.159,A 0.000,B 0.000,C 90.000,E1 64.588} C_DIS
LIN {X 0.125,Y -570.852,Z 891.151,A 0.000,B 0.000,C 90.000,E1 63.204} C_DIS
LIN {X 0.049,Y -570.661,Z 891.144,A 0.000,B 0.000,C 90.000,E1 61.847} C_DIS
LIN {X 0.182,Y -570.292,Z 891.133,A 0.000,B 0.000,C 90.000,E1 59.921} C_DIS
LIN {X -0.112,Y -569.647,Z 891.125,A 0.000,B 0.000,C 90.000,E1 58.584} C_DIS
LIN {X 0.244,Y -569.124,Z 891.119,A 0.000,B 0.000,C 90.000,E1 57.454} C_DIS
LIN {X 0.341,Y -567.890,Z 891.110,A 0.000,B 0.000,C 90.000,E1 55.801} C_DIS
LIN {X -0.173,Y -566.619,Z 891.103,A 0.000,B 0.000,C 90.000,E1 54.482} C_DIS
LIN {X 0.069,Y -564.873,Z 891.095,A 0.000,B 0.000,C 90.000,E1 53.084} C_DIS
LIN {X -0.050,Y -563.747,Z 891.090,A 0.000,B 0.000,C 90.000,E1 52.271} C_DIS
LIN {X -0.174,Y -562.448,Z 891.086,A 0.000,B 0.000,C 90.000,E1 51.457} C_DIS
LIN {X -0.211,Y -560.430,Z 891.080,A 0.000,B 0.000,C 90.000,E1 50.356} C_DIS
LIN {X -0.029,Y -559.313,Z 891.077,A 0.000,B 0.000,C 90.000,E1 49.784} C_DIS
LIN {X 0.160,Y -557.341,Z 891.072,A 0.000,B 0.000,C 90.000,E1 48.933} C_DIS
LIN {X -0.107,Y -555.893,Z 891.069,A 0.000,B 0.000,C 90.000,E1 48.405} C_DIS
LIN {X 0.051,Y -553.382,Z 891.064,A 0.000,B 0.000,C 90.000,E1 47.553} C_DIS
LIN {X 0.178,Y -550.560,Z 891.060,A 0.000,B 0.000,C 90.000,E1 46.701} C_DIS
LIN {X 0.240,Y -548.587,Z 891.057,A 0.000,B 0.000,C 90.000,E1 46.134} C_DIS
LIN {X -0.079,Y -545.315,Z 891.052,A 0.000,B 0.000,C 90.000,E1 45.324} C_DIS
LIN {X 0.146,Y -542.315,Z 891.048,A 0.000,B 0.000,C 90.000,E1 44.595} C_DIS
LIN {X 0.148,Y -539.687,Z 891.045,A 0.000,B 0.000,C 90.000,E1 44.028} C_DIS
LIN {X 0.128,Y -536.814,Z 891.042,A 0.000,B 0.000,C 90.000,E1 43.461} C_DIS
LIN {X -0.103,Y -532.835,Z 891.038,A 0.000,B 0.000,C 90.000,E1 42.771} C_DIS
LIN {X -0.174,Y -529.447,Z 891.034,A 0.000,B 0.000,C 90.000,E1 42.204} C_DIS
LIN {X 0.119,Y -525.905,Z 891.031,A 0.000,B 0.000,C 90.000,E1 41.595} C_DIS
LIN {X 0.233,Y -523.115,Z 891.029,A 0.000,B 0.000,C 90.000,E1 41.148} C_DIS
LIN {X 0.023,Y -517.029,Z 891.024,A 0.000,B 0.000,C 90.000,E1 40.297} C_DIS
LIN {X 0.016,Y -511.620,Z 891.020,A 0.000,B 0.000,C 90.000,E1 39.564} C_DIS
LIN {X 0.135,Y -507.226,Z 891.017,A 0.000,B 0.000,C 90.000,E1 38.991} C_DIS
LIN {X -0.194,Y -501.100,Z 891.013,A 0.000,B 0.000,C 90.000,E1 38.302} C_DIS
LIN {X 0.201,Y -497.050,Z 891.010,A 0.000,B 0.000,C 90.000,E1 37.810} C_DIS
LIN {X -0.240,Y -490.323,Z 891.006,A 0.000,B 0.000,C 90.000,E1 37.156} C_DIS
LIN {X 0.020,Y -483.249,Z 891.002,A 0.000,B 0.000,C 90.000,E1 36.423} C_DIS
LIN {X -0.040,Y -477.333,Z 890.999,A 0.000,B 0.000,C 90.000,E1 35.884} C_DIS
LIN {X 0.131,Y -466.809,Z 890.994,A 0.000,B 0.000,C 90.000,E1 34.945} C_DIS
LIN {X 0.257,Y -454.554,Z 890.989,A 0.000,B 0.000,C 90.000,E1 33.913} C_DIS
LIN {X -0.153,Y -443.632,Z 890.984,A 0.000,B 0.000,C 90.000,E1 33.086} C_DIS
LIN {X 0.156,Y -419.220,Z 890.972,A 0.000,B 0.000,C 90.000,E1 31.003} C_DIS
LIN {X -0.206,Y -404.376,Z 890.965,A 0.000,B 0.000,C 90.000,E1 29.667} C_DIS
LIN {X -0.063,Y -398.815,Z 890.962,A 0.000,B 0.000,C 90.000,E1 29.077} C_DIS
LIN {X -0.130,Y -396.491,Z 890.960,A 0.000,B 0.000,C 90.000,E1 28.821} C_DIS
LIN {X 0.038,Y -393.402,Z 890.958,A 0.000,B 0.000,C 90.000,E1 28.359} C_DIS
LIN {X -0.077,Y -392.598,Z 890.957,A 0.000,B 0.000,C 90.000,E1 28.231} C_DIS
LIN {X -0.099,Y -391.357,Z 890.955,A 0.000,B 0.000,C 90.000,E1 27.897} C_DIS
LIN {X 0.135,Y -390.353,Z 890.954,A 0.000,B 0.000,C 90.000,E1 27.641} C_DIS
LIN {X -0.047,Y -389.204,Z 890.950,A 0.000,B 0.000,C 90.000,E1 27.001} C_DIS
LIN {X -0.017,Y -388.931,Z 890.947,A 0.000,B 0.000,C 90.000,E1 26.437} C_DIS
LIN {X 0.191,Y -389.160,Z 890.941,A 0.000,B 0.000,C 90.000,E1 25.335} C_DIS
LIN {X -0.014,Y -391.441,Z 890.925,A 0.000,B 0.000,C 90.000,E1 22.514} C_DIS
LIN {X -0.028,Y -394.667,Z 890.907,A 0.000,B 0.000,C 90.000,E1 19.322} C_DIS
LIN {X -0.080,Y -397.514,Z 890.894,A 0.000,B 0.000,C 90.000,E1 16.858} C_DIS
LIN {X 0.171,Y -399.764,Z 890.884,A 0.000,B 0.000,C 90.000,E1 15.064} C_DIS
LIN {X -0.068,Y -404.051,Z 890.866,A 0.000,B 0.000,C 90.000,E1 11.951} C_DIS
LIN {X 0.078,Y -408.286,Z 890.851,A 0.000,B 0.000,C 90.000,E1 9.151} C_DIS
LIN {X -0.184,Y -412.958,Z 890.836,A 0.000,B 0.000,C 90.000,E1 6.429} C_DIS
LIN {X -0.082,Y -416.762,Z 890.824,A 0.000,B 0.000,C 90.000,E1 4.359} C_DIS
LIN {X 0.064,Y -420.195,Z 890.815,A 0.000,B 0.000,C 90.000,E1 2.636} C_DIS
LIN {X -0.207,Y -427.403,Z 890.797,A 0.000,B 0.000,C 90.000,E1 359.484} C_DIS
LIN {X 0.139,Y -431.517,Z 890.788,A 0.000,B 0.000,C 90.000,E1 357.764} C_DIS
LIN {X 0.049,Y -434.971,Z 890.780,A 0.000,B 0.000,C 90.000,E1 356.445} C_DIS
LIN {X -0.180,Y -437.140,Z 890.777,A 0.000,B 0.000,C 90.000,E1 355.812} C_DIS
LIN {X -0.007,Y -439.224,Z 890.774,A 0.000,B 0.000,C 90.000,E1 355.298} C_DIS
LIN {X 0.190,Y -441.198,Z 890.772,A 0.000,B 0.000,C 90.000,E1 354.951} C_DIS
LIN {X -0.141,Y -442.344,Z 890.771,A 0.000,B 0.000,C 90.000,E1 354.837} C_DIS
LIN {X -0.023,Y -443.238,Z 890.771,A 0.000,B 0.000,C 90.000,E1 354.723} C_DIS
LIN {X 0.172,Y -445.981,Z 890.770,A 0.000,B 0.000,C 90.000,E1 354.489} C_DIS
LIN {X 0.193,Y -449.248,Z 890.768,A 0.000,B 0.000,C 90.000,E1 354.261} C_DIS
LIN {X 0.141,Y -455.538,Z 890.767,A 0.000,B 0.000,C 90.000,E1 353.970} C_DIS
LIN {X 0.172,Y -467.156,Z 890.764,A 0.000,B 0.000,C 90.000,E1 353.457} C_DIS
LIN {X -0.244,Y -475.587,Z 890.762,A 0.000,B 0.000,C 90.000,E1 353.109} C_DIS
LIN {X 0.211,Y -485.590,Z 890.759,A 0.000,B 0.000,C 90.000,E1 352.534} C_DIS
LIN {X 0.049,Y -495.311,Z 890.756,A 0.000,B 0.000,C 90.000,E1 352.008} C_DIS
LIN {X 0.104,Y -504.949,Z 890.753,A 0.000,B 0.000,C 90.000,E1 351.432} C_DIS
LIN {X 0.126,Y -515.971,Z 890.749,A 0.000,B 0.000,C 90.000,E1 350.735} C_DIS
LIN {X 0.211,Y -523.507,Z 890.746,A 0.000,B 0.000,C 90.000,E1 350.218} C_DIS
LIN {X 0.025,Y -531.028,Z 890.743,A 0.000,B 0.000,C 90.000,E1 349.690} C_DIS
LIN {X -0.012,Y -539.658,Z 890.739,A 0.000,B 0.000,C 90.000,E1 348.993} C_DIS
LIN {X -0.164,Y -545.265,Z 890.736,A 0.000,B 0.000,C 90.000,E1 348.522} C_DIS
LIN {X 0.114,Y -551.816,Z 890.733,A 0.000,B 0.000,C 90.000,E1 347.881} C_DIS
LIN {X 0.165,Y -556.969,Z 890.730,A 0.000,B 0.000,C 90.000,E1 347.353} C_DIS
LIN {X 0.238,Y -561.828,Z 890.727,A 0.000,B 0.000,C 90.000,E1 346.825} C_DIS
LIN {X 0.307,Y -568.995,Z 890.722,A 0.000,B 0.000,C 90.000,E1 345.992} C_DIS
LIN {X 0.115,Y -573.411,Z 890.719,A 0.000,B 0.000,C 90.000,E1 345.463} C_DIS
LIN {X -0.152,Y -578.624,Z 890.716,A 0.000,B 0.000,C 90.000,E1 344.810} C_DIS
LIN {X 0.093,Y -584.472,Z 890.711,A 0.000,B 0.000,C 90.000,E1 343.976} C_DIS
LIN {X -0.084,Y -589.013,Z 890.707,A 0.000,B 0.000,C 90.000,E1 343.323} C_DIS
LIN {X 0.144,Y -595.606,Z 890.701,A 0.000,B 0.000,C 90.000,E1 342.236} C_DIS
LIN {X 0.000,Y -600.166,Z 890.697,A 0.000,B 0.000,C 90.000,E1 341.456} C_DIS
LIN {X -0.144,Y -605.218,Z 890.692,A 0.000,B 0.000,C 90.000,E1 340.550} C_DIS
LIN {X -0.295,Y -611.294,Z 890.685,A 0.000,B 0.000,C 90.000,E1 339.390} C_DIS
LIN {X -0.116,Y -616.400,Z 890.680,A 0.000,B 0.000,C 90.000,E1 338.337} C_DIS
LIN {X -0.099,Y -621.209,Z 890.674,A 0.000,B 0.000,C 90.000,E1 337.305} C_DIS
LIN {X -0.118,Y -625.741,Z 890.668,A 0.000,B 0.000,C 90.000,E1 336.282} C_DIS
LIN {X 0.253,Y -629.956,Z 890.663,A 0.000,B 0.000,C 90.000,E1 335.229} C_DIS
LIN {X 0.133,Y -634.786,Z 890.656,A 0.000,B 0.000,C 90.000,E1 333.973} C_DIS
LIN {X -0.256,Y -638.373,Z 890.650,A 0.000,B 0.000,C 90.000,E1 332.999} C_DIS
LIN {X -0.028,Y -641.739,Z 890.644,A 0.000,B 0.000,C 90.000,E1 331.975} C_DIS
LIN {X -0.014,Y -644.790,Z 890.639,A 0.000,B 0.000,C 90.000,E1 330.973} C_DIS
LIN {X 0.220,Y -649.124,Z 890.630,A 0.000,B 0.000,C 90.000,E1 329.459} C_DIS
LIN {X -0.119,Y -652.494,Z 890.624,A 0.000,B 0.000,C 90.000,E1 328.250} C_DIS
LIN {X -0.047,Y -654.347,Z 890.620,A 0.000,B 0.000,C 90.000,E1 327.502} C_DIS
LIN {X -0.315,Y -657.075,Z 890.613,A 0.000,B 0.000,C 90.000,E1 326.294} C_DIS
LIN {X -0.186,Y -659.357,Z 890.606,A 0.000,B 0.000,C 90.000,E1 325.055} C_DIS
LIN {X -0.218,Y -660.548,Z 890.602,A 0.000,B 0.000,C 90.000,E1 324.322} C_DIS
LIN {X -0.133,Y -661.968,Z 890.596,A 0.000,B 0.000,C 90.000,E1 323.336} C_DIS
LIN {X 0.010,Y -663.629,Z 890.588,A 0.000,B 0.000,C 90.000,E1 321.859} C_DIS
LIN {X -0.013,Y -664.904,Z 890.581,A 0.000,B 0.000,C 90.000,E1 320.642} C_DIS
LIN {X 0.064,Y -666.405,Z 890.573,A 0.000,B 0.000,C 90.000,E1 319.175} C_DIS
LIN {X 0.098,Y -668.463,Z 890.563,A 0.000,B 0.000,C 90.000,E1 317.229} C_DIS
LIN {X -0.328,Y -669.756,Z 890.556,A 0.000,B 0.000,C 90.000,E1 316.053} C_DIS
LIN {X -0.269,Y -670.942,Z 890.549,A 0.000,B 0.000,C 90.000,E1 314.838} C_DIS
LIN {X -0.207,Y -671.826,Z 890.544,A 0.000,B 0.000,C 90.000,E1 313.866} C_DIS
LIN {X 0.369,Y -673.089,Z 890.537,A 0.000,B 0.000,C 90.000,E1 312.609} C_DIS
LIN {X 0.011,Y -674.237,Z 890.530,A 0.000,B 0.000,C 90.000,E1 311.434} C_DIS
LIN {X 0.287,Y -675.668,Z 890.521,A 0.000,B 0.000,C 90.000,E1 309.725} C_DIS
LIN {X 0.055,Y -676.858,Z 890.513,A 0.000,B 0.000,C 90.000,E1 308.302} C_DIS
LIN {X -0.047,Y -677.892,Z 890.505,A 0.000,B 0.000,C 90.000,E1 306.870} C_DIS
LIN {X -0.129,Y -678.731,Z 890.498,A 0.000,B 0.000,C 90.000,E1 305.678} C_DIS
LIN {X -0.030,Y -679.672,Z 890.489,A 0.000,B 0.000,C 90.000,E1 303.992} C_DIS
LIN {X -0.112,Y -680.884,Z 890.478,A 0.000,B 0.000,C 90.000,E1 302.084} C_DIS
LIN {X 0.413,Y -682.379,Z 890.468,A 0.000,B 0.000,C 90.000,E1 300.129} C_DIS
LIN {X 0.111,Y -684.757,Z 890.454,A 0.000,B 0.000,C 90.000,E1 297.769} C_DIS
LIN {X 0.336,Y -687.023,Z 890.444,A 0.000,B 0.000,C 90.000,E1 295.848} C_DIS
LIN {X -0.076,Y -688.441,Z 890.437,A 0.000,B 0.000,C 90.000,E1 294.695} C_DIS
LIN {X -0.129,Y -689.496,Z 890.431,A 0.000,B 0.000,C 90.000,E1 293.515} C_DIS
LIN {X 0.285,Y -689.219,Z 890.427,A 0.000,B 0.000,C 90.000,E1 292.770} C_DIS
LIN {X -0.164,Y -688.098,Z 890.424,A 0.000,B 0.000,C 90.000,E1 292.333} C_DIS
LIN {X 0.058,Y -687.262,Z 890.423,A 0.000,B 0.000,C 90.000,E1 292.078} C_DIS
LIN {X -0.091,Y -686.513,Z 890.422,A 0.000,B 0.000,C 90.000,E1 291.972} C_DIS
LIN {X 0.082,Y -682.003,Z 890.419,A 0.000,B 0.000,C 90.000,E1 291.482} C_DIS
LIN {X 0.184,Y -680.599,Z 890.419,A 0.000,B 0.000,C 90.000,E1 291.354} C_DIS
LIN {X -0.242,Y -678.597,Z 890.418,A 0.000,B 0.000,C 90.000,E1 291.280} C_DIS
LIN {X -0.140,Y -668.540,Z 890.416,A 0.000,B 0.000,C 90.000,E1 290.918} C_DIS
LIN {X 0.080,Y -662.928,Z 890.415,A 0.000,B 0.000,C 90.000,E1 290.737} C_DIS
LIN {X 0.116,Y -661.509,Z 890.415,A 0.000,B 0.000,C 90.000,E1 290.684} C_DIS
LIN {X 0.300,Y -657.812,Z 890.414,A 0.000,B 0.000,C 90.000,E1 290.482} C_DIS
LIN {X 0.246,Y -657.732,Z 890.414,A 0.000,B 0.000,C 90.000,E1 290.482} C_DIS
LIN {X 0.220,Y -657.014,Z 890.413,A 0.000,B 0.000,C 90.000,E1 290.375} C_DIS
LIN {X 0.176,Y -657.004,Z 890.413,A 0.000,B 0.000,C 90.000,E1 290.375} C_DIS
LIN {X 0.104,Y -656.919,Z 890.412,A 0.000,B 0.000,C 90.000,E1 290.174} C_DIS
LIN {X -0.056,Y -658.150,Z 890.410,A 0.000,B 0.000,C 90.000,E1 289.758} C_DIS
LIN {X -0.021,Y -660.890,Z 890.406,A 0.000,B 0.000,C 90.000,E1 289.141} C_DIS
LIN {X 0.136,Y -665.906,Z 890.401,A 0.000,B 0.000,C 90.000,E1 288.181} C_DIS
LIN {X 0.023,Y -668.972,Z 890.398,A 0.000,B 0.000,C 90.000,E1 287.583} C_DIS
LIN {X 0.067,Y -671.284,Z 890.395,A 0.000,B 0.000,C 90.000,E1 287.094} C_DIS
LIN {X -0.134,Y -674.160,Z 890.391,A 0.000,B 0.000,C 90.000,E1 286.386} C_DIS
LIN {X -0.064,Y -675.782,Z 890.388,A 0.000,B 0.000,C 90.000,E1 285.898} C_DIS
LIN {X -0.218,Y -677.686,Z 890.384,A 0.000,B 0.000,C 90.000,E1 285.190} C_DIS
LIN {X -0.351,Y -679.269,Z 890.380,A 0.000,B 0.000,C 90.000,E1 284.481} C_DIS
LIN {X 0.160,Y -681.020,Z 890.375,A 0.000,B 0.000,C 90.000,E1 283.480} C_DIS
LIN {X 0.030,Y -682.261,Z 890.370,A 0.000,B 0.000,C 90.000,E1 282.535} C_DIS
LIN {X -0.063,Y -682.853,Z 890.366,A 0.000,B 0.000,C 90.000,E1 281.827} C_DIS
LIN {X -0.261,Y -683.014,Z 890.363,A 0.000,B 0.000,C 90.000,E1 281.366} C_DIS
LIN {X 0.317,Y -682.703,Z 890.359,A 0.000,B 0.000,C 90.000,E1 280.602} C_DIS
LIN {X 0.128,Y -682.268,Z 890.356,A 0.000,B 0.000,C 90.000,E1 280.141} C_DIS
LIN {X 0.056,Y -681.447,Z 890.354,A 0.000,B 0.000,C 90.000,E1 279.670} C_DIS
LIN {X -0.138,Y -680.328,Z 890.351,A 0.000,B 0.000,C 90.000,E1 279.208} C_DIS
LIN {X -0.333,Y -678.897,Z 890.349,A 0.000,B 0.000,C 90.000,E1 278.746} C_DIS
LIN {X 0.234,Y -677.195,Z 890.346,A 0.000,B 0.000,C 90.000,E1 278.219} C_DIS
LIN {X 0.082,Y -676.316,Z 890.344,A 0.000,B 0.000,C 90.000,E1 277.992} C_DIS
LIN {X -0.204,Y -672.952,Z 890.340,A 0.000,B 0.000,C 90.000,E1 277.296} C_DIS
LIN {X 0.225,Y -670.447,Z 890.338,A 0.000,B 0.000,C 90.000,E1 276.777} C_DIS
LIN {X -0.118,Y -666.910,Z 890.334,A 0.000,B 0.000,C 90.000,E1 276.201} C_DIS
LIN {X -0.307,Y -664.653,Z 890.332,A 0.000,B 0.000,C 90.000,E1 275.853} C_DIS
LIN {X 0.058,Y -661.176,Z 890.330,A 0.000,B 0.000,C 90.000,E1 275.334} C_DIS
LIN {X 0.297,Y -656.168,Z 890.326,A 0.000,B 0.000,C 90.000,E1 274.702} C_DIS
LIN {X -0.103,Y -651.666,Z 890.324,A 0.000,B 0.000,C 90.000,E1 274.245} C_DIS
LIN {X 0.167,Y -645.494,Z 890.320,A 0.000,B 0.000,C 90.000,E1 273.612} C_DIS
LIN {X 0.047,Y -638.860,Z 890.317,A 0.000,B 0.000,C 90.000,E1 273.037} C_DIS
LIN {X 0.158,Y -631.867,Z 890.314,A 0.000,B 0.000,C 90.000,E1 272.465} C_DIS
LIN {X -0.302,Y -624.681,Z 890.311,A 0.000,B 0.000,C 90.000,E1 272.007} C_DIS
LIN {X 0.140,Y -616.764,Z 890.308,A 0.000,B 0.000,C 90.000,E1 271.489} C_DIS
LIN {X 0.017,Y -610.157,Z 890.306,A 0.000,B 0.000,C 90.000,E1 271.146} C_DIS
LIN {X 0.271,Y -603.309,Z 890.305,A 0.000,B 0.000,C 90.000,E1 270.802} C_DIS
LIN {X -0.282,Y -598.102,Z 890.303,A 0.000,B 0.000,C 90.000,E1 270.630} C_DIS
LIN {X -0.026,Y -592.602,Z 890.302,A 0.000,B 0.000,C 90.000,E1 270.401} C_DIS
LIN {X -0.144,Y -585.438,Z 890.301,A 0.000,B 0.000,C 90.000,E1 270.172} C_DIS
LIN {X 0.123,Y -578.091,Z 890.300,A 0.000,B 0.000,C 90.000,E1 269.943} C_DIS
LIN {X -0.053,Y -571.632,Z 890.299,A 0.000,B 0.000,C 90.000,E1 269.828} C_DIS
LIN {X 0.173,Y -564.792,Z 890.299,A 0.000,B 0.000,C 90.000,E1 269.714} C_DIS
LIN {X -0.231,Y -552.337,Z 890.298,A 0.000,B 0.000,C 90.000,E1 269.656} C_DIS
LIN {X -0.110,Y -549.328,Z 890.297,A 0.000,B 0.000,C 90.000,E1 269.542} C_DIS
LIN {X -0.040,Y -547.073,Z 890.296,A 0.000,B 0.000,C 90.000,E1 269.312} C_DIS
LIN {X -0.088,Y -546.671,Z 890.296,A 0.000,B 0.000,C 90.000,E1 269.255} C_DIS
LIN {X -0.092,Y -545.458,Z 890.294,A 0.000,B 0.000,C 90.000,E1 268.912} C_DIS
LIN {X -0.180,Y -544.543,Z 890.291,A 0.000,B 0.000,C 90.000,E1 268.453} C_DIS
LIN {X 0.084,Y -542.393,Z 890.280,A 0.000,B 0.000,C 90.000,E1 266.445} C_DIS
LIN {X -0.184,Y -540.814,Z 890.268,A 0.000,B 0.000,C 90.000,E1 264.204} C_DIS
LIN {X -0.044,Y -540.072,Z 890.261,A 0.000,B 0.000,C 90.000,E1 263.053} C_DIS
LIN {X 0.150,Y -539.104,Z 890.255,A 0.000,B 0.000,C 90.000,E1 261.894} C_DIS
LIN {X -0.132,Y -537.708,Z 890.247,A 0.000,B 0.000,C 90.000,E1 260.500} C_DIS
LIN {X 0.204,Y -535.643,Z 890.236,A 0.000,B 0.000,C 90.000,E1 258.465} C_DIS
LIN {X -0.047,Y -534.077,Z 890.228,A 0.000,B 0.000,C 90.000,E1 257.061} C_DIS
LIN {X -0.249,Y -532.592,Z 890.222,A 0.000,B 0.000,C 90.000,E1 255.936} C_DIS
LIN {X -0.227,Y -530.079,Z 890.211,A 0.000,B 0.000,C 90.000,E1 253.921} C_DIS
LIN {X -0.145,Y -527.991,Z 890.201,A 0.000,B 0.000,C 90.000,E1 252.181} C_DIS
LIN {X 0.212,Y -526.926,Z 890.196,A 0.000,B 0.000,C 90.000,E1 251.275} C_DIS
LIN {X -0.274,Y -525.128,Z 890.188,A 0.000,B 0.000,C 90.000,E1 249.880} C_DIS
LIN {X 0.040,Y -522.728,Z 890.178,A 0.000,B 0.000,C 90.000,E1 248.103} C_DIS
LIN {X 0.185,Y -521.068,Z 890.172,A 0.000,B 0.000,C 90.000,E1 246.922} C_DIS
LIN {X -0.169,Y -519.324,Z 890.165,A 0.000,B 0.000,C 90.000,E1 245.793} C_DIS
LIN {X -0.060,Y -516.651,Z 890.156,A 0.000,B 0.000,C 90.000,E1 244.024} C_DIS
LIN {X 0.096,Y -514.238,Z 890.148,A 0.000,B 0.000,C 90.000,E1 242.538} C_DIS
LIN {X 0.206,Y -511.675,Z 890.139,A 0.000,B 0.000,C 90.000,E1 241.051} C_DIS
LIN {X 0.039,Y -508.014,Z 890.128,A 0.000,B 0.000,C 90.000,E1 238.997} C_DIS
LIN {X -0.167,Y -505.404,Z 890.120,A 0.000,B 0.000,C 90.000,E1 237.533} C_DIS
LIN {X 0.233,Y -503.036,Z 890.113,A 0.000,B 0.000,C 90.000,E1 236.294} C_DIS
LIN {X 0.183,Y -500.375,Z 890.106,A 0.000,B 0.000,C 90.000,E1 235.102} C_DIS
LIN {X -0.164,Y -496.163,Z 890.096,A 0.000,B 0.000,C 90.000,E1 233.336} C_DIS
LIN {X -0.160,Y -492.814,Z 890.088,A 0.000,B 0.000,C 90.000,E1 231.823} C_DIS
LIN {X 0.083,Y -489.337,Z 890.079,A 0.000,B 0.000,C 90.000,E1 230.275} C_DIS
LIN {X 0.057,Y -486.612,Z 890.073,A 0.000,B 0.000,C 90.000,E1 229.057} C_DIS
LIN {X -0.150,Y -484.545,Z 890.068,A 0.000,B 0.000,C 90.000,E1 228.162} C_DIS
LIN {X 0.134,Y -479.745,Z 890.056,A 0.000,B 0.000,C 90.000,E1 225.972} C_DIS
LIN {X 0.165,Y -475.536,Z 890.045,A 0.000,B 0.000,C 90.000,E1 224.109} C_DIS
LIN {X 0.117,Y -471.298,Z 890.035,A 0.000,B 0.000,C 90.000,E1 222.243} C_DIS
LIN {X -0.100,Y -467.793,Z 890.026,A 0.000,B 0.000,C 90.000,E1 220.701} C_DIS
LIN {X -0.034,Y -464.429,Z 890.017,A 0.000,B 0.000,C 90.000,E1 219.116} C_DIS
LIN {X 0.033,Y -461.083,Z 890.009,A 0.000,B 0.000,C 90.000,E1 217.523} C_DIS
LIN {X 0.140,Y -457.021,Z 889.998,A 0.000,B 0.000,C 90.000,E1 215.598} C_DIS
LIN {X -0.116,Y -452.962,Z 889.987,A 0.000,B 0.000,C 90.000,E1 213.706} C_DIS
LIN {X 0.120,Y -448.142,Z 889.975,A 0.000,B 0.000,C 90.000,E1 211.416} C_DIS
LIN {X -0.002,Y -443.164,Z 889.962,A 0.000,B 0.000,C 90.000,E1 209.155} C_DIS
LIN {X 0.035,Y -439.571,Z 889.953,A 0.000,B 0.000,C 90.000,E1 207.513} C_DIS
LIN {X 0.011,Y -435.202,Z 889.942,A 0.000,B 0.000,C 90.000,E1 205.540} C_DIS
LIN {X 0.069,Y -432.405,Z 889.935,A 0.000,B 0.000,C 90.000,E1 204.207} C_DIS
LIN {X -0.107,Y -427.416,Z 889.922,A 0.000,B 0.000,C 90.000,E1 201.897} C_DIS
LIN {X -0.108,Y -424.643,Z 889.914,A 0.000,B 0.000,C 90.000,E1 200.556} C_DIS
LIN {X -0.189,Y -420.532,Z 889.903,A 0.000,B 0.000,C 90.000,E1 198.544} C_DIS
LIN {X 0.133,Y -417.090,Z 889.893,A 0.000,B 0.000,C 90.000,E1 196.804} C_DIS
LIN {X 0.172,Y -411.601,Z 889.878,A 0.000,B 0.000,C 90.000,E1 194.064} C_DIS
LIN {X 0.106,Y -407.659,Z 889.867,A 0.000,B 0.000,C 90.000,E1 192.007} C_DIS
LIN {X -0.152,Y -404.971,Z 889.859,A 0.000,B 0.000,C 90.000,E1 190.658} C_DIS
LIN {X -0.139,Y -400.736,Z 889.848,A 0.000,B 0.000,C 90.000,E1 188.568} C_DIS
LIN {X 0.035,Y -395.886,Z 889.834,A 0.000,B 0.000,C 90.000,E1 186.087} C_DIS
LIN {X 0.114,Y -392.147,Z 889.822,A 0.000,B 0.000,C 90.000,E1 183.955} C_DIS
LIN {X -0.052,Y -388.221,Z 889.808,A 0.000,B 0.000,C 90.000,E1 181.489} C_DIS
LIN {X -0.039,Y -386.153,Z 889.800,A 0.000,B 0.000,C 90.000,E1 180.057} C_DIS
LIN {X 0.118,Y -382.842,Z 889.788,A 0.000,B 0.000,C 90.000,E1 177.879} C_DIS
LIN {X 0.174,Y -381.171,Z 889.782,A 0.000,B 0.000,C 90.000,E1 176.788} C_DIS
LIN {X -0.138,Y -376.633,Z 889.764,A 0.000,B 0.000,C 90.000,E1 173.571} C_DIS
LIN {X 0.178,Y -375.345,Z 889.756,A 0.000,B 0.000,C 90.000,E1 172.064} C_DIS
LIN {X 0.163,Y -374.974,Z 889.750,A 0.000,B 0.000,C 90.000,E1 170.971} C_DIS
LIN {X 0.172,Y -375.437,Z 889.743,A 0.000,B 0.000,C 90.000,E1 169.690} C_DIS
LIN {X 0.106,Y -376.076,Z 889.741,A 0.000,B 0.000,C 90.000,E1 169.285} C_DIS
LIN {X 0.067,Y -376.509,Z 889.739,A 0.000,B 0.000,C 90.000,E1 168.926} C_DIS
LIN {X -0.041,Y -377.461,Z 889.737,A 0.000,B 0.000,C 90.000,E1 168.578} C_DIS
LIN {X -0.160,Y -378.630,Z 889.734,A 0.000,B 0.000,C 90.000,E1 168.049} C_DIS
LIN {X 0.118,Y -379.197,Z 889.732,A 0.000,B 0.000,C 90.000,E1 167.825} C_DIS
LIN {X -0.070,Y -381.205,Z 889.730,A 0.000,B 0.000,C 90.000,E1 167.409} C_DIS
LIN {X 0.106,Y -385.132,Z 889.727,A 0.000,B 0.000,C 90.000,E1 166.769} C_DIS
LIN {X 0.105,Y -386.514,Z 889.726,A 0.000,B 0.000,C 90.000,E1 166.589} C_DIS
LIN {X -0.145,Y -391.610,Z 889.723,A 0.000,B 0.000,C 90.000,E1 166.117} C_DIS
LIN {X -0.132,Y -403.630,Z 889.719,A 0.000,B 0.000,C 90.000,E1 165.338} C_DIS
LIN {X -0.150,Y -410.862,Z 889.716,A 0.000,B 0.000,C 90.000,E1 164.936} C_DIS
LIN {X 0.091,Y -415.737,Z 889.715,A 0.000,B 0.000,C 90.000,E1 164.629} C_DIS
LIN {X 0.201,Y -422.125,Z 889.712,A 0.000,B 0.000,C 90.000,E1 164.212} C_DIS
LIN {X 0.046,Y -430.186,Z 889.709,A 0.000,B 0.000,C 90.000,E1 163.685} C_DIS
LIN {X 0.254,Y -436.490,Z 889.707,A 0.000,B 0.000,C 90.000,E1 163.196} C_DIS
LIN {X 0.019,Y -444.111,Z 889.703,A 0.000,B 0.000,C 90.000,E1 162.598} C_DIS
LIN {X 0.199,Y -450.085,Z 889.701,A 0.000,B 0.000,C 90.000,E1 162.054} C_DIS
LIN {X 0.119,Y -455.987,Z 889.698,A 0.000,B 0.000,C 90.000,E1 161.529} C_DIS
LIN {X -0.041,Y -463.237,Z 889.694,A 0.000,B 0.000,C 90.000,E1 160.859} C_DIS
LIN {X -0.081,Y -468.809,Z 889.691,A 0.000,B 0.000,C 90.000,E1 160.296} C_DIS
LIN {X -0.105,Y -475.764,Z 889.686,A 0.000,B 0.000,C 90.000,E1 159.571} C_DIS
LIN {X -0.086,Y -482.308,Z 889.682,A 0.000,B 0.000,C 90.000,E1 158.827} C_DIS
LIN {X 0.033,Y -490.943,Z 889.676,A 0.000,B 0.000,C 90.000,E1 157.741} C_DIS
LIN {X -0.060,Y -500.188,Z 889.670,A 0.000,B 0.000,C 90.000,E1 156.538} C_DIS
LIN {X -0.111,Y -505.587,Z 889.666,A 0.000,B 0.000,C 90.000,E1 155.793} C_DIS
LIN {X -0.083,Y -511.995,Z 889.661,A 0.000,B 0.000,C 90.000,E1 154.897} C_DIS
LIN {X 0.292,Y -522.031,Z 889.652,A 0.000,B 0.000,C 90.000,E1 153.384} C_DIS
LIN {X 0.052,Y -530.687,Z 889.645,A 0.000,B 0.000,C 90.000,E1 152.103} C_DIS
LIN {X 0.180,Y -534.210,Z 889.642,A 0.000,B 0.000,C 90.000,E1 151.513} C_DIS
LIN {X 0.117,Y -543.426,Z 889.633,A 0.000,B 0.000,C 90.000,E1 149.950} C_DIS
LIN {X -0.233,Y -548.809,Z 889.628,A 0.000,B 0.000,C 90.000,E1 148.997} C_DIS
LIN {X 0.077,Y -553.382,Z 889.623,A 0.000,B 0.000,C 90.000,E1 148.122} C_DIS
LIN {X -0.283,Y -561.560,Z 889.615,A 0.000,B 0.000,C 90.000,E1 146.628} C_DIS
LIN {X -0.301,Y -567.765,Z 889.608,A 0.000,B 0.000,C 90.000,E1 145.388} C_DIS
LIN {X 0.109,Y -573.683,Z 889.601,A 0.000,B 0.000,C 90.000,E1 144.116} C_DIS
LIN {X -0.004,Y -578.162,Z 889.595,A 0.000,B 0.000,C 90.000,E1 143.176} C_DIS
LIN {X 0.025,Y -584.285,Z 889.588,A 0.000,B 0.000,C 90.000,E1 141.823} C_DIS
LIN {X 0.060,Y -590.245,Z 889.581,A 0.000,B 0.000,C 90.000,E1 140.481} C_DIS
LIN {X -0.161,Y -593.775,Z 889.576,A 0.000,B 0.000,C 90.000,E1 139.703} C_DIS
LIN {X 0.197,Y -600.709,Z 889.567,A 0.000,B 0.000,C 90.000,E1 138.081} C_DIS
LIN {X 0.056,Y -606.645,Z 889.560,A 0.000,B 0.000,C 90.000,E1 136.782} C_DIS
LIN {X -0.191,Y -613.743,Z 889.551,A 0.000,B 0.000,C 90.000,E1 135.243} C_DIS
LIN {X 0.019,Y -618.372,Z 889.546,A 0.000,B 0.000,C 90.000,E1 134.190} C_DIS
LIN {X -0.427,Y -625.062,Z 889.537,A 0.000,B 0.000,C 90.000,E1 132.690} C_DIS
LIN {X -0.157,Y -630.444,Z 889.530,A 0.000,B 0.000,C 90.000,E1 131.391} C_DIS
LIN {X 0.207,Y -635.680,Z 889.523,A 0.000,B 0.000,C 90.000,E1 130.092} C_DIS
LIN {X -0.039,Y -638.762,Z 889.519,A 0.000,B 0.000,C 90.000,E1 129.358} C_DIS
LIN {X -0.048,Y -644.512,Z 889.510,A 0.000,B 0.000,C 90.000,E1 127.855} C_DIS
LIN {X 0.249,Y -649.302,Z 889.503,A 0.000,B 0.000,C 90.000,E1 126.583} C_DIS
LIN {X 0.187,Y -652.911,Z 889.498,A 0.000,B 0.000,C 90.000,E1 125.598} C_DIS
LIN {X -0.281,Y -657.131,Z 889.491,A 0.000,B 0.000,C 90.000,E1 124.405} C_DIS
LIN {X 0.303,Y -660.304,Z 889.486,A 0.000,B 0.000,C 90.000,E1 123.372} C_DIS
LIN {X 0.334,Y -661.835,Z 889.483,A 0.000,B 0.000,C 90.000,E1 122.880} C_DIS
LIN {X 0.192,Y -665.123,Z 889.476,A 0.000,B 0.000,C 90.000,E1 121.671} C_DIS
LIN {X 0.385,Y -666.803,Z 889.472,A 0.000,B 0.000,C 90.000,E1 120.924} C_DIS
LIN {X -0.017,Y -669.163,Z 889.465,A 0.000,B 0.000,C 90.000,E1 119.745} C_DIS
LIN {X 0.367,Y -670.744,Z 889.460,A 0.000,B 0.000,C 90.000,E1 118.743} C_DIS
LIN {X 0.058,Y -673.226,Z 889.451,A 0.000,B 0.000,C 90.000,E1 117.078} C_DIS
LIN {X 0.169,Y -674.237,Z 889.445,A 0.000,B 0.000,C 90.000,E1 116.104} C_DIS
LIN {X -0.008,Y -674.930,Z 889.440,A 0.000,B 0.000,C 90.000,E1 115.155} C_DIS
LIN {X -0.358,Y -675.166,Z 889.436,A 0.000,B 0.000,C 90.000,E1 114.463} C_DIS
LIN {X 0.004,Y -675.108,Z 889.433,A 0.000,B 0.000,C 90.000,E1 113.951} C_DIS
LIN {X 0.093,Y -674.796,Z 889.430,A 0.000,B 0.000,C 90.000,E1 113.462} C_DIS
LIN {X -0.172,Y -673.847,Z 889.428,A 0.000,B 0.000,C 90.000,E1 113.003} C_DIS
LIN {X -0.260,Y -673.154,Z 889.426,A 0.000,B 0.000,C 90.000,E1 112.770} C_DIS
LIN {X -0.005,Y -671.025,Z 889.424,A 0.000,B 0.000,C 90.000,E1 112.386} C_DIS
LIN {X -0.096,Y -669.279,Z 889.423,A 0.000,B 0.000,C 90.000,E1 112.153} C_DIS
LIN {X -0.016,Y -668.136,Z 889.422,A 0.000,B 0.000,C 90.000,E1 112.025} C_DIS
LIN {X 0.238,Y -661.357,Z 889.420,A 0.000,B 0.000,C 90.000,E1 111.535} C_DIS
LIN {X -0.067,Y -659.282,Z 889.419,A 0.000,B 0.000,C 90.000,E1 111.461} C_DIS
LIN {X 0.214,Y -654.981,Z 889.418,A 0.000,B 0.000,C 90.000,E1 111.280} C_DIS
LIN {X 0.065,Y -644.870,Z 889.417,A 0.000,B 0.000,C 90.000,E1 111.046} C_DIS
LIN {X 0.098,Y -635.919,Z 889.416,A 0.000,B 0.000,C 90.000,E1 110.865} C_DIS
LIN {X 0.051,Y -623.014,Z 889.414,A 0.000,B 0.000,C 90.000,E1 110.556} C_DIS
LIN {X 0.085,Y -616.770,Z 889.413,A 0.000,B 0.000,C 90.000,E1 110.375} C_DIS
LIN {X 0.048,Y -610.840,Z 889.412,A 0.000,B 0.000,C 90.000,E1 110.174} C_DIS
LIN {X -0.080,Y -602.310,Z 889.410,A 0.000,B 0.000,C 90.000,E1 109.812} C_DIS
LIN {X -0.330,Y -590.319,Z 889.407,A 0.000,B 0.000,C 90.000,E1 109.214} C_DIS
LIN {X -0.189,Y -586.994,Z 889.406,A 0.000,B 0.000,C 90.000,E1 109.033} C_DIS
LIN {X 0.224,Y -580.467,Z 889.404,A 0.000,B 0.000,C 90.000,E1 108.671} C_DIS
LIN {X -0.191,Y -569.707,Z 889.402,A 0.000,B 0.000,C 90.000,E1 108.308} C_DIS
LIN {X -0.063,Y -563.047,Z 889.400,A 0.000,B 0.000,C 90.000,E1 108.055} C_DIS
LIN {X -0.154,Y -558.707,Z 889.399,A 0.000,B 0.000,C 90.000,E1 107.819} C_DIS
LIN {X -0.086,Y -557.252,Z 889.398,A 0.000,B 0.000,C 90.000,E1 107.583} C_DIS
LIN {X 0.229,Y -556.609,Z 889.396,A 0.000,B 0.000,C 90.000,E1 107.221} C_DIS
LIN {X -0.244,Y -556.388,Z 889.393,A 0.000,B 0.000,C 90.000,E1 106.677} C_DIS
LIN {X 0.281,Y -557.238,Z 889.379,A 0.000,B 0.000,C 90.000,E1 104.120} C_DIS
LIN {X -0.100,Y -558.600,Z 889.365,A 0.000,B 0.000,C 90.000,E1 101.658} C_DIS
LIN {X -0.187,Y -559.998,Z 889.354,A 0.000,B 0.000,C 90.000,E1 99.726} C_DIS
LIN {X -0.181,Y -560.986,Z 889.346,A 0.000,B 0.000,C 90.000,E1 98.341} C_DIS
LIN {X 0.005,Y -561.993,Z 889.337,A 0.000,B 0.000,C 90.000,E1 96.663} C_DIS
LIN {X -0.092,Y -562.612,Z 889.331,A 0.000,B 0.000,C 90.000,E1 95.568} C_DIS
LIN {X -0.087,Y -563.296,Z 889.323,A 0.000,B 0.000,C 90.000,E1 94.188} C_DIS
LIN {X -0.078,Y -563.816,Z 889.316,A 0.000,B 0.000,C 90.000,E1 92.808} C_DIS
LIN {X 0.012,Y -564.410,Z 889.306,A 0.000,B 0.000,C 90.000,E1 91.146} C_DIS
LIN {X -0.115,Y -564.663,Z 889.300,A 0.000,B 0.000,C 90.000,E1 90.057} C_DIS
LIN {X -0.239,Y -564.945,Z 889.294,A 0.000,B 0.000,C 90.000,E1 88.969} C_DIS
LIN {X -0.124,Y -565.266,Z 889.285,A 0.000,B 0.000,C 90.000,E1 87.306} C_DIS
LIN {X 0.131,Y -565.562,Z 889.274,A 0.000,B 0.000,C 90.000,E1 85.355} C_DIS
LIN {X 0.029,Y -565.979,Z 889.262,A 0.000,B 0.000,C 90.000,E1 83.166} C_DIS
LIN {X -0.249,Y -566.366,Z 889.253,A 0.000,B 0.000,C 90.000,E1 81.546} C_DIS
LIN {X 0.208,Y -567.030,Z 889.242,A 0.000,B 0.000,C 90.000,E1 79.577} C_DIS
LIN {X -0.230,Y -567.908,Z 889.232,A 0.000,B 0.000,C 90.000,E1 77.701} C_DIS
LIN {X -0.135,Y -568.650,Z 889.222,A 0.000,B 0.000,C 90.000,E1 76.047} C_DIS
LIN {X 0.025,Y -569.144,Z 889.216,A 0.000,B 0.000,C 90.000,E1 74.936} C_DIS
LIN {X -0.220,Y -569.614,Z 889.210,A 0.000,B 0.000,C 90.000,E1 73.866} C_DIS
LIN {X 0.250,Y -569.894,Z 889.204,A 0.000,B 0.000,C 90.000,E1 72.725} C_DIS
LIN {X -0.191,Y -570.322,Z 889.197,A 0.000,B 0.000,C 90.000,E1 71.402} C_DIS
LIN {X -0.090,Y -570.612,Z 889.188,A 0.000,B 0.000,C 90.000,E1 69.752} C_DIS
LIN {X 0.017,Y -570.812,Z 889.178,A 0.000,B 0.000,C 90.000,E1 68.103} C_DIS
LIN {X -0.193,Y -570.915,Z 889.169,A 0.000,B 0.000,C 90.000,E1 66.485} C_DIS
LIN {X -0.168,Y -570.948,Z 889.160,A 0.000,B 0.000,C 90.000,E1 64.845} C_DIS
LIN {X -0.149,Y -570.872,Z 889.151,A 0.000,B 0.000,C 90.000,E1 63.204} C_DIS
LIN {X -0.226,Y -570.647,Z 889.143,A 0.000,B 0.000,C 90.000,E1 61.847} C_DIS
LIN {X -0.203,Y -570.294,Z 889.134,A 0.000,B 0.000,C 90.000,E1 60.205} C_DIS
LIN {X -0.266,Y -570.154,Z 889.131,A 0.000,B 0.000,C 90.000,E1 59.665} C_DIS
LIN {X 0.153,Y -569.174,Z 889.121,A 0.000,B 0.000,C 90.000,E1 57.709} C_DIS
LIN {X 0.140,Y -568.184,Z 889.113,A 0.000,B 0.000,C 90.000,E1 56.342} C_DIS
LIN {X -0.018,Y -567.221,Z 889.107,A 0.000,B 0.000,C 90.000,E1 55.261} C_DIS
LIN {X 0.337,Y -566.427,Z 889.102,A 0.000,B 0.000,C 90.000,E1 54.402} C_DIS
LIN {X 0.012,Y -565.028,Z 889.096,A 0.000,B 0.000,C 90.000,E1 53.336} C_DIS
LIN {X -0.334,Y -563.480,Z 889.090,A 0.000,B 0.000,C 90.000,E1 52.271} C_DIS
LIN {X -0.020,Y -562.154,Z 889.086,A 0.000,B 0.000,C 90.000,E1 51.412} C_DIS
LIN {X -0.163,Y -560.641,Z 889.081,A 0.000,B 0.000,C 90.000,E1 50.598} C_DIS
LIN {X 0.041,Y -558.932,Z 889.076,A 0.000,B 0.000,C 90.000,E1 49.747} C_DIS
LIN {X -0.213,Y -557.644,Z 889.073,A 0.000,B 0.000,C 90.000,E1 49.218} C_DIS
LIN {X -0.034,Y -555.448,Z 889.069,A 0.000,B 0.000,C 90.000,E1 48.366} C_DIS
LIN {X -0.249,Y -552.844,Z 889.064,A 0.000,B 0.000,C 90.000,E1 47.553} C_DIS
LIN {X -0.125,Y -549.999,Z 889.059,A 0.000,B 0.000,C 90.000,E1 46.701} C_DIS
LIN {X 0.344,Y -546.890,Z 889.055,A 0.000,B 0.000,C 90.000,E1 45.810} C_DIS
LIN {X -0.002,Y -544.644,Z 889.052,A 0.000,B 0.000,C 90.000,E1 45.283} C_DIS
LIN {X 0.018,Y -542.227,Z 889.048,A 0.000,B 0.000,C 90.000,E1 44.717} C_DIS
LIN {X -0.174,Y -538.875,Z 889.045,A 0.000,B 0.000,C 90.000,E1 44.028} C_DIS
LIN {X -0.197,Y -535.952,Z 889.041,A 0.000,B 0.000,C 90.000,E1 43.461} C_DIS
LIN {X 0.145,Y -532.752,Z 889.038,A 0.000,B 0.000,C 90.000,E1 42.852} C_DIS
LIN {X -0.117,Y -528.450,Z 889.034,A 0.000,B 0.000,C 90.000,E1 42.162} C_DIS
LIN {X -0.068,Y -523.915,Z 889.030,A 0.000,B 0.000,C 90.000,E1 41.434} C_DIS
LIN {X 0.038,Y -520.947,Z 889.028,A 0.000,B 0.000,C 90.000,E1 40.987} C_DIS
LIN {X 0.199,Y -514.755,Z 889.023,A 0.000,B 0.000,C 90.000,E1 40.092} C_DIS
LIN {X 0.050,Y -510.254,Z 889.020,A 0.000,B 0.000,C 90.000,E1 39.519} C_DIS
LIN {X 0.194,Y -505.442,Z 889.016,A 0.000,B 0.000,C 90.000,E1 38.910} C_DIS
LIN {X -0.249,Y -500.520,Z 889.013,A 0.000,B 0.000,C 90.000,E1 38.382} C_DIS
LIN {X 0.310,Y -495.092,Z 889.010,A 0.000,B 0.000,C 90.000,E1 37.729} C_DIS
LIN {X -0.182,Y -488.169,Z 889.006,A 0.000,B 0.000,C 90.000,E1 37.076} C_DIS
LIN {X -0.055,Y -482.467,Z 889.003,A 0.000,B 0.000,C 90.000,E1 36.503} C_DIS
LIN {X -0.078,Y -475.243,Z 888.999,A 0.000,B 0.000,C 90.000,E1 35.851} C_DIS
LIN {X 0.303,Y -466.221,Z 888.995,A 0.000,B 0.000,C 90.000,E1 35.025} C_DIS
LIN {X -0.096,Y -454.133,Z 888.989,A 0.000,B 0.000,C 90.000,E1 34.072} C_DIS
LIN {X -0.110,Y -440.218,Z 888.983,A 0.000,B 0.000,C 90.000,E1 32.959} C_DIS
LIN {X -0.008,Y -417.244,Z 888.972,A 0.000,B 0.000,C 90.000,E1 31.003} C_DIS
LIN {X 0.054,Y -403.910,Z 888.965,A 0.000,B 0.000,C 90.000,E1 29.745} C_DIS
LIN {X -0.038,Y -398.121,Z 888.962,A 0.000,B 0.000,C 90.000,E1 29.155} C_DIS
LIN {X 0.059,Y -395.458,Z 888.960,A 0.000,B 0.000,C 90.000,E1 28.821} C_DIS
LIN {X -0.218,Y -394.239,Z 888.959,A 0.000,B 0.000,C 90.000,E1 28.693} C_DIS
LIN {X -0.039,Y -391.957,Z 888.957,A 0.000,B 0.000,C 90.000,E1 28.281} C_DIS
LIN {X 0.163,Y -390.681,Z 888.955,A 0.000,B 0.000,C 90.000,E1 27.897} C_DIS
LIN {X -0.175,Y -390.212,Z 888.954,A 0.000,B 0.000,C 90.000,E1 27.769} C_DIS
LIN {X 0.003,Y -389.267,Z 888.951,A 0.000,B 0.000,C 90.000,E1 27.206} C_DIS
LIN {X 0.034,Y -388.971,Z 888.947,A 0.000,B 0.000,C 90.000,E1 26.488} C_DIS
LIN {X 0.074,Y -389.256,Z 888.941,A 0.000,B 0.000,C 90.000,E1 25.412} C_DIS
LIN {X 0.071,Y -391.837,Z 888.923,A 0.000,B 0.000,C 90.000,E1 22.206} C_DIS
LIN {X -0.119,Y -394.742,Z 888.908,A 0.000,B 0.000,C 90.000,E1 19.396} C_DIS
LIN {X -0.043,Y -397.582,Z 888.894,A 0.000,B 0.000,C 90.000,E1 16.913} C_DIS
LIN {X 0.180,Y -400.280,Z 888.882,A 0.000,B 0.000,C 90.000,E1 14.773} C_DIS
LIN {X -0.035,Y -404.583,Z 888.865,A 0.000,B 0.000,C 90.000,E1 11.658} C_DIS
LIN {X 0.107,Y -408.310,Z 888.851,A 0.000,B 0.000,C 90.000,E1 9.208} C_DIS
LIN {X -0.155,Y -412.972,Z 888.836,A 0.000,B 0.000,C 90.000,E1 6.486} C_DIS
LIN {X 0.002,Y -418.152,Z 888.821,A 0.000,B 0.000,C 90.000,E1 3.726} C_DIS
LIN {X -0.090,Y -424.631,Z 888.804,A 0.000,B 0.000,C 90.000,E1 0.688} C_DIS
LIN {X -0.016,Y -429.972,Z 888.791,A 0.000,B 0.000,C 90.000,E1 358.453} C_DIS
LIN {X 0.140,Y -436.015,Z 888.779,A 0.000,B 0.000,C 90.000,E1 356.102} C_DIS
LIN {X -0.128,Y -437.653,Z 888.776,A 0.000,B 0.000,C 90.000,E1 355.641} C_DIS
LIN {X -0.034,Y -439.015,Z 888.774,A 0.000,B 0.000,C 90.000,E1 355.298} C_DIS
LIN {X -0.021,Y -442.141,Z 888.771,A 0.000,B 0.000,C 90.000,E1 354.780} C_DIS
LIN {X 0.032,Y -443.441,Z 888.770,A 0.000,B 0.000,C 90.000,E1 354.609} C_DIS
LIN {X 0.105,Y -445.527,Z 888.769,A 0.000,B 0.000,C 90.000,E1 354.432} C_DIS
LIN {X 0.059,Y -448.783,Z 888.768,A 0.000,B 0.000,C 90.000,E1 354.204} C_DIS
LIN {X -0.155,Y -456.738,Z 888.766,A 0.000,B 0.000,C 90.000,E1 353.856} C_DIS
LIN {X -0.096,Y -467.079,Z 888.763,A 0.000,B 0.000,C 90.000,E1 353.394} C_DIS
LIN {X 0.169,Y -473.714,Z 888.762,A 0.000,B 0.000,C 90.000,E1 353.053} C_DIS
LIN {X -0.240,Y -483.666,Z 888.759,A 0.000,B 0.000,C 90.000,E1 352.591} C_DIS
LIN {X 0.209,Y -493.208,Z 888.756,A 0.000,B 0.000,C 90.000,E1 352.008} C_DIS
LIN {X -0.073,Y -504.528,Z 888.752,A 0.000,B 0.000,C 90.000,E1 351.376} C_DIS
LIN {X -0.127,Y -515.688,Z 888.748,A 0.000,B 0.000,C 90.000,E1 350.679} C_DIS
LIN {X -0.089,Y -523.345,Z 888.745,A 0.000,B 0.000,C 90.000,E1 350.151} C_DIS
LIN {X 0.160,Y -530.825,Z 888.742,A 0.000,B 0.000,C 90.000,E1 349.577} C_DIS
LIN {X 0.208,Y -539.558,Z 888.738,A 0.000,B 0.000,C 90.000,E1 348.870} C_DIS
LIN {X -0.062,Y -545.136,Z 888.736,A 0.000,B 0.000,C 90.000,E1 348.409} C_DIS
LIN {X -0.186,Y -550.375,Z 888.733,A 0.000,B 0.000,C 90.000,E1 347.937} C_DIS
LIN {X 0.092,Y -554.405,Z 888.731,A 0.000,B 0.000,C 90.000,E1 347.521} C_DIS
LIN {X -0.176,Y -560.716,Z 888.727,A 0.000,B 0.000,C 90.000,E1 346.881} C_DIS
LIN {X 0.016,Y -566.800,Z 888.723,A 0.000,B 0.000,C 90.000,E1 346.172} C_DIS
LIN {X 0.063,Y -570.296,Z 888.721,A 0.000,B 0.000,C 90.000,E1 345.755} C_DIS
LIN {X -0.122,Y -574.678,Z 888.718,A 0.000,B 0.000,C 90.000,E1 345.227} C_DIS
LIN {X -0.130,Y -578.827,Z 888.715,A 0.000,B 0.000,C 90.000,E1 344.685} C_DIS
LIN {X 0.209,Y -583.703,Z 888.711,A 0.000,B 0.000,C 90.000,E1 343.976} C_DIS
LIN {X -0.050,Y -589.236,Z 888.707,A 0.000,B 0.000,C 90.000,E1 343.196} C_DIS
LIN {X -0.059,Y -596.596,Z 888.700,A 0.000,B 0.000,C 90.000,E1 342.000} C_DIS
LIN {X 0.047,Y -600.380,Z 888.696,A 0.000,B 0.000,C 90.000,E1 341.329} C_DIS
LIN {X -0.093,Y -605.449,Z 888.691,A 0.000,B 0.000,C 90.000,E1 340.423} C_DIS
LIN {X -0.236,Y -611.515,Z 888.685,A 0.000,B 0.000,C 90.000,E1 339.263} C_DIS
LIN {X -0.279,Y -616.634,Z 888.679,A 0.000,B 0.000,C 90.000,E1 338.230} C_DIS
LIN {X -0.022,Y -620.876,Z 888.674,A 0.000,B 0.000,C 90.000,E1 337.305} C_DIS
LIN {X -0.295,Y -625.446,Z 888.668,A 0.000,B 0.000,C 90.000,E1 336.305} C_DIS
LIN {X 0.346,Y -630.706,Z 888.661,A 0.000,B 0.000,C 90.000,E1 334.973} C_DIS
LIN {X 0.201,Y -634.613,Z 888.656,A 0.000,B 0.000,C 90.000,E1 333.973} C_DIS
LIN {X -0.191,Y -638.208,Z 888.650,A 0.000,B 0.000,C 90.000,E1 332.999} C_DIS
LIN {X 0.037,Y -641.594,Z 888.644,A 0.000,B 0.000,C 90.000,E1 331.975} C_DIS
LIN {X 0.049,Y -644.715,Z 888.639,A 0.000,B 0.000,C 90.000,E1 330.973} C_DIS
LIN {X 0.282,Y -649.093,Z 888.630,A 0.000,B 0.000,C 90.000,E1 329.459} C_DIS
LIN {X -0.058,Y -652.495,Z 888.624,A 0.000,B 0.000,C 90.000,E1 328.250} C_DIS
LIN {X 0.014,Y -654.382,Z 888.620,A 0.000,B 0.000,C 90.000,E1 327.502} C_DIS
LIN {X -0.252,Y -657.122,Z 888.613,A 0.000,B 0.000,C 90.000,E1 326.294} C_DIS
LIN {X -0.217,Y -659.036,Z 888.607,A 0.000,B 0.000,C 90.000,E1 325.308} C_DIS
LIN {X -0.151,Y -660.673,Z 888.602,A 0.000,B 0.000,C 90.000,E1 324.322} C_DIS
LIN {X -0.066,Y -662.106,Z 888.596,A 0.000,B 0.000,C 90.000,E1 323.336} C_DIS
LIN {X -0.002,Y -663.584,Z 888.590,A 0.000,B 0.000,C 90.000,E1 322.110} C_DIS
LIN {X 0.080,Y -664.904,Z 888.583,A 0.000,B 0.000,C 90.000,E1 320.884} C_DIS
LIN {X 0.135,Y -666.906,Z 888.572,A 0.000,B 0.000,C 90.000,E1 318.933} C_DIS
LIN {X 0.188,Y -668.988,Z 888.561,A 0.000,B 0.000,C 90.000,E1 316.986} C_DIS
LIN {X -0.217,Y -670.478,Z 888.553,A 0.000,B 0.000,C 90.000,E1 315.567} C_DIS
LIN {X -0.176,Y -671.185,Z 888.549,A 0.000,B 0.000,C 90.000,E1 314.838} C_DIS
LIN {X -0.128,Y -671.905,Z 888.545,A 0.000,B 0.000,C 90.000,E1 314.109} C_DIS
LIN {X 0.036,Y -673.600,Z 888.536,A 0.000,B 0.000,C 90.000,E1 312.405} C_DIS
LIN {X -0.309,Y -674.708,Z 888.529,A 0.000,B 0.000,C 90.000,E1 311.229} C_DIS
LIN {X -0.013,Y -676.160,Z 888.520,A 0.000,B 0.000,C 90.000,E1 309.519} C_DIS
LIN {X 0.173,Y -677.131,Z 888.513,A 0.000,B 0.000,C 90.000,E1 308.302} C_DIS
LIN {X 0.077,Y -678.195,Z 888.505,A 0.000,B 0.000,C 90.000,E1 306.870} C_DIS
LIN {X 0.000,Y -679.018,Z 888.498,A 0.000,B 0.000,C 90.000,E1 305.678} C_DIS
LIN {X -0.067,Y -679.851,Z 888.490,A 0.000,B 0.000,C 90.000,E1 304.246} C_DIS
LIN {X -0.156,Y -681.063,Z 888.480,A 0.000,B 0.000,C 90.000,E1 302.339} C_DIS
LIN {X -0.183,Y -682.316,Z 888.470,A 0.000,B 0.000,C 90.000,E1 300.669} C_DIS
LIN {X 0.024,Y -684.032,Z 888.460,A 0.000,B 0.000,C 90.000,E1 298.743} C_DIS
LIN {X -0.383,Y -686.156,Z 888.449,A 0.000,B 0.000,C 90.000,E1 296.873} C_DIS
LIN {X 0.271,Y -688.182,Z 888.440,A 0.000,B 0.000,C 90.000,E1 295.155} C_DIS
LIN {X -0.127,Y -689.328,Z 888.433,A 0.000,B 0.000,C 90.000,E1 294.003} C_DIS
LIN {X 0.052,Y -689.707,Z 888.431,A 0.000,B 0.000,C 90.000,E1 293.515} C_DIS
LIN {X 0.240,Y -689.587,Z 888.428,A 0.000,B 0.000,C 90.000,E1 293.025} C_DIS
LIN {X -0.167,Y -689.451,Z 888.427,A 0.000,B 0.000,C 90.000,E1 292.823} C_DIS
LIN {X -0.205,Y -688.928,Z 888.425,A 0.000,B 0.000,C 90.000,E1 292.589} C_DIS
LIN {X 0.243,Y -687.439,Z 888.423,A 0.000,B 0.000,C 90.000,E1 292.078} C_DIS
LIN {X 0.095,Y -686.737,Z 888.422,A 0.000,B 0.000,C 90.000,E1 291.972} C_DIS
LIN {X -0.219,Y -683.394,Z 888.420,A 0.000,B 0.000,C 90.000,E1 291.642} C_DIS
LIN {X -0.264,Y -680.685,Z 888.419,A 0.000,B 0.000,C 90.000,E1 291.408} C_DIS
LIN {X -0.067,Y -678.787,Z 888.418,A 0.000,B 0.000,C 90.000,E1 291.280} C_DIS
LIN {X 0.078,Y -668.571,Z 888.416,A 0.000,B 0.000,C 90.000,E1 290.918} C_DIS
LIN {X -0.277,Y -661.338,Z 888.415,A 0.000,B 0.000,C 90.000,E1 290.737} C_DIS
LIN {X 0.330,Y -657.313,Z 888.414,A 0.000,B 0.000,C 90.000,E1 290.482} C_DIS
LIN {X 0.273,Y -657.217,Z 888.414,A 0.000,B 0.000,C 90.000,E1 290.482} C_DIS
LIN {X -0.319,Y -656.528,Z 888.413,A 0.000,B 0.000,C 90.000,E1 290.429} C_DIS
LIN {X -0.369,Y -656.513,Z 888.413,A 0.000,B 0.000,C 90.000,E1 290.429} C_DIS
LIN {X -0.155,Y -656.410,Z 888.412,A 0.000,B 0.000,C 90.000,E1 290.174} C_DIS
LIN {X -0.318,Y -657.692,Z 888.410,A 0.000,B 0.000,C 90.000,E1 289.758} C_DIS
LIN {X 0.337,Y -660.477,Z 888.406,A 0.000,B 0.000,C 90.000,E1 289.087} C_DIS
LIN {X -0.060,Y -664.944,Z 888.402,A 0.000,B 0.000,C 90.000,E1 288.290} C_DIS
LIN {X -0.243,Y -667.460,Z 888.399,A 0.000,B 0.000,C 90.000,E1 287.819} C_DIS
LIN {X -0.287,Y -670.915,Z 888.395,A 0.000,B 0.000,C 90.000,E1 287.094} C_DIS
LIN {X 0.216,Y -672.883,Z 888.392,A 0.000,B 0.000,C 90.000,E1 286.567} C_DIS
LIN {X 0.223,Y -675.402,Z 888.388,A 0.000,B 0.000,C 90.000,E1 285.843} C_DIS
LIN {X 0.069,Y -677.272,Z 888.384,A 0.000,B 0.000,C 90.000,E1 285.134} C_DIS
LIN {X -0.022,Y -678.380,Z 888.381,A 0.000,B 0.000,C 90.000,E1 284.662} C_DIS
LIN {X -0.021,Y -680.166,Z 888.376,A 0.000,B 0.000,C 90.000,E1 283.703} C_DIS
LIN {X -0.288,Y -681.226,Z 888.372,A 0.000,B 0.000,C 90.000,E1 283.008} C_DIS
LIN {X 0.279,Y -681.996,Z 888.368,A 0.000,B 0.000,C 90.000,E1 282.243} C_DIS
LIN {X 0.214,Y -682.334,Z 888.366,A 0.000,B 0.000,C 90.000,E1 281.771} C_DIS
LIN {X 0.149,Y -682.498,Z 888.363,A 0.000,B 0.000,C 90.000,E1 281.299} C_DIS
LIN {X -0.082,Y -682.133,Z 888.359,A 0.000,B 0.000,C 90.000,E1 280.602} C_DIS
LIN {X -0.274,Y -681.665,Z 888.356,A 0.000,B 0.000,C 90.000,E1 280.141} C_DIS
LIN {X 0.321,Y -680.845,Z 888.354,A 0.000,B 0.000,C 90.000,E1 279.613} C_DIS
LIN {X 0.126,Y -679.722,Z 888.351,A 0.000,B 0.000,C 90.000,E1 279.151} C_DIS
LIN {X 0.029,Y -678.253,Z 888.348,A 0.000,B 0.000,C 90.000,E1 278.681} C_DIS
LIN {X -0.334,Y -675.647,Z 888.344,A 0.000,B 0.000,C 90.000,E1 277.992} C_DIS
LIN {X 0.114,Y -673.455,Z 888.342,A 0.000,B 0.000,C 90.000,E1 277.473} C_DIS
LIN {X -0.117,Y -670.404,Z 888.338,A 0.000,B 0.000,C 90.000,E1 276.891} C_DIS
LIN {X 0.205,Y -666.902,Z 888.335,A 0.000,B 0.000,C 90.000,E1 276.258} C_DIS
LIN {X -0.074,Y -663.838,Z 888.332,A 0.000,B 0.000,C 90.000,E1 275.796} C_DIS
LIN {X 0.284,Y -660.320,Z 888.330,A 0.000,B 0.000,C 90.000,E1 275.277} C_DIS
LIN {X -0.095,Y -656.309,Z 888.327,A 0.000,B 0.000,C 90.000,E1 274.821} C_DIS
LIN {X 0.107,Y -650.633,Z 888.323,A 0.000,B 0.000,C 90.000,E1 274.188} C_DIS
LIN {X -0.226,Y -644.420,Z 888.320,A 0.000,B 0.000,C 90.000,E1 273.612} C_DIS
LIN {X -0.287,Y -637.783,Z 888.317,A 0.000,B 0.000,C 90.000,E1 273.037} C_DIS
LIN {X -0.113,Y -630.796,Z 888.314,A 0.000,B 0.000,C 90.000,E1 272.465} C_DIS
LIN {X -0.295,Y -624.690,Z 888.311,A 0.000,B 0.000,C 90.000,E1 272.064} C_DIS
LIN {X 0.123,Y -616.736,Z 888.309,A 0.000,B 0.000,C 90.000,E1 271.547} C_DIS
LIN {X 0.006,Y -610.197,Z 888.307,A 0.000,B 0.000,C 90.000,E1 271.203} C_DIS
LIN {X 0.084,Y -601.551,Z 888.305,A 0.000,B 0.000,C 90.000,E1 270.802} C_DIS
LIN {X 0.214,Y -596.360,Z 888.303,A 0.000,B 0.000,C 90.000,E1 270.573} C_DIS
LIN {X -0.048,Y -590.941,Z 888.302,A 0.000,B 0.000,C 90.000,E1 270.401} C_DIS
LIN {X -0.073,Y -583.604,Z 888.301,A 0.000,B 0.000,C 90.000,E1 270.172} C_DIS
LIN {X 0.061,Y -577.694,Z 888.300,A 0.000,B 0.000,C 90.000,E1 270.000} C_DIS
LIN {X 0.000,Y -571.640,Z 888.299,A 0.000,B 0.000,C 90.000,E1 269.885} C_DIS
LIN {X 0.193,Y -564.259,Z 888.299,A 0.000,B 0.000,C 90.000,E1 269.771} C_DIS
LIN {X -0.146,Y -552.216,Z 888.298,A 0.000,B 0.000,C 90.000,E1 269.714} C_DIS
LIN {X 0.167,Y -549.619,Z 888.298,A 0.000,B 0.000,C 90.000,E1 269.599} C_DIS
LIN {X -0.189,Y -546.648,Z 888.296,A 0.000,B 0.000,C 90.000,E1 269.370} C_DIS
LIN {X -0.227,Y -546.615,Z 888.296,A 0.000,B 0.000,C 90.000,E1 269.370} C_DIS
LIN {X 0.215,Y -545.636,Z 888.295,A 0.000,B 0.000,C 90.000,E1 269.026} C_DIS
LIN {X -0.150,Y -544.605,Z 888.292,A 0.000,B 0.000,C 90.000,E1 268.511} C_DIS
LIN {X 0.115,Y -542.509,Z 888.281,A 0.000,B 0.000,C 90.000,E1 266.502} C_DIS
LIN {X -0.148,Y -540.925,Z 888.268,A 0.000,B 0.000,C 90.000,E1 264.261} C_DIS
LIN {X -0.005,Y -540.188,Z 888.262,A 0.000,B 0.000,C 90.000,E1 263.109} C_DIS
LIN {X 0.192,Y -539.244,Z 888.255,A 0.000,B 0.000,C 90.000,E1 261.951} C_DIS
LIN {X -0.086,Y -537.848,Z 888.248,A 0.000,B 0.000,C 90.000,E1 260.557} C_DIS
LIN {X 0.257,Y -535.775,Z 888.236,A 0.000,B 0.000,C 90.000,E1 258.522} C_DIS
LIN {X 0.011,Y -534.215,Z 888.228,A 0.000,B 0.000,C 90.000,E1 257.117} C_DIS
LIN {X -0.143,Y -532.384,Z 888.221,A 0.000,B 0.000,C 90.000,E1 255.700} C_DIS
LIN {X -0.129,Y -529.878,Z 888.209,A 0.000,B 0.000,C 90.000,E1 253.685} C_DIS
LIN {X -0.054,Y -527.816,Z 888.200,A 0.000,B 0.000,C 90.000,E1 251.945} C_DIS
LIN {X 0.140,Y -525.614,Z 888.190,A 0.000,B 0.000,C 90.000,E1 250.188} C_DIS
LIN {X -0.030,Y -524.487,Z 888.185,A 0.000,B 0.000,C 90.000,E1 249.337} C_DIS
LIN {X 0.138,Y -522.881,Z 888.179,A 0.000,B 0.000,C 90.000,E1 248.156} C_DIS
LIN {X -0.240,Y -520.804,Z 888.171,A 0.000,B 0.000,C 90.000,E1 246.741} C_DIS
LIN {X 0.087,Y -519.026,Z 888.164,A 0.000,B 0.000,C 90.000,E1 245.537} C_DIS
